// TwinCAT 3 PLC project Nepionic_Motion
// Title: Nepionic_Motion
// Company: Nepionic
// Author: Nepionic
// ProjectVersion: 0.1.0
// ProgramVersion: 3.1.4026.19
// libraries:
//   Nepionic_Core, * (Nepionic)
//   Tc2_MC2, * (Beckhoff Automation GmbH)
//   Tc2_MC2_Drive, * (Beckhoff Automation GmbH)
// project tree:
//   Builders/Homing/ HomeBuilder.TcIO, PositionHomeBuilder.TcIO
//   Builders/Homing/Implementation/ DefaultPositionHomeBuilder.TcPOU, DefaultHomeBuilder.TcPOU, DefaultHomeBuilderParameters.TcDUT
//   Builders/Motion/ GearInBuilder.TcIO (not stored), MotionBuilder.TcIO, AbsoluteMoveBuilder.TcIO, MoveBuilder.TcIO, RelativeMoveBuilder.TcIO, VelocityMoveBuilder.TcIO
//   Builders/Motion/Implementation/ DefaultMotionBuilderParameters.TcDUT, DefaultGearInBuilder.TcPOU, DefaultMotionBuilder.TcPOU, DefaultAbsoluteMoveBuilder.TcPOU, DefaultMoveBuilder.TcPOU, DefaultRelativeMoveBuilder.TcPOU, DefaultVelocityMoveBuilder.TcPOU
//   Commands/Administrative/ ResetCommand.TcPOU (not stored)
//   Commands/Homing/ HomeCommand.TcPOU
//   Commands/SoE/ ResetSoeDriveCommand.TcPOU
//   Commands/Coupling/ GearInCommand.TcPOU, GearOutCommand.TcPOU (not stored)
//   Commands/PointToPoint/ MoveAbsoluteCommand.TcPOU, MoveAdditiveCommand.TcPOU, MoveContinuousAbsoluteCommand.TcPOU, MoveContinuousRelativeCommand.TcPOU, MoveModuloCommand.TcPOU, MoveRelativeCommand.TcPOU, MoveVelocityCommand.TcPOU
//   Commands/Stops/ HaltCommand.TcPOU, StopCommand.TcPOU
//   Command/ Mc2Command.TcPOU, Mc2MotionCommand.TcPOU, MotionCommand.TcIO
//   Functions/ Mc2BufferModeConvertFrom.TcPOU, Mc2BufferModeConvertTo.TcPOU, Mc2DirectionConvertFrom.TcPOU, Mc2DirectionConvertTo.TcPOU, Mc2EncoderReferenceModeConvertFrom.TcPOU, Mc2EncoderReferenceModeConvertTo.TcPOU, Mc2HomingModeConvertFrom.TcPOU, Mc2HomingModeConvertTo.TcPOU
//   Axis/ Axis.TcIO, Mc2Axis.TcPOU
//   Types/ AxisMotionState.TcDUT (not stored), EncoderReferenceMode.TcDUT, HomingMode.TcDUT, MotionBufferMode.TcDUT, MotionDirection.TcDUT

// ---- Builders/Homing/Implementation/DefaultHomeBuilderParameters.TcDUT
TYPE DefaultHomeBuilderParameters :
STRUCT
	position : LREAL;
	homing_mode : HomingMode;
	reference_mode : EncoderReferenceMode;
	search_direction : MotionDirection;
	search_velocity : LREAL;
	sync_direction : MotionDirection;
	sync_velocity : LREAL;
	buffer_mode : MotionBufferMode;
END_STRUCT
END_TYPE

// ---- Builders/Motion/Implementation/DefaultMotionBuilderParameters.TcDUT
TYPE DefaultMotionBuilderParameters :
STRUCT
	position : LREAL;
	distance : LREAL;
	velocity : LREAL;
	acceleration : LREAL;
	deceleration : LREAL;
	jerk : LREAL;
	buffer_mode : MotionBufferMode;
	ratio_numerator : LREAL;
	ratio_denominator : UINT;
END_STRUCT
END_TYPE

// ---- Types/EncoderReferenceMode.TcDUT
{attribute 'qualified_only'}
{attribute 'strict'}
{attribute 'to_string'}
TYPE EncoderReferenceMode :
(
    Default := TO_INT(EncoderReferenceMode_Default),
    PlcCam := TO_INT(EncoderReferenceMode_PlcCam),
    HardwareSync := TO_INT(EncoderReferenceMode_HardwareSync),
    HardwareLatchPositive := TO_INT(EncoderReferenceMode_HardwareLatchPos),
    HardwareLatchNegative := TO_INT(EncoderReferenceMode_HardwareLatchNeg),
    SoftwareSync := TO_INT(EncoderReferenceMode_SoftwareSync),
    SoftDriveLatchPositive := TO_INT(EncoderReferenceMode_SoftDriveLatchPos),
    SoftDriveLatchNegative := TO_INT(EncoderReferenceMode_SoftDriveLatchNeg)
);
END_TYPE

// ---- Types/HomingMode.TcDUT
{attribute 'qualified_only'}
{attribute 'strict'}
{attribute 'to_string'}
TYPE HomingMode :
(
	Default := TO_INT(Tc2_Mc2.MC_DefaultHoming),
	Direct := TO_INT(Tc2_Mc2.MC_Direct),
	ForceCalibration := TO_INT(Tc2_Mc2.MC_ForceCalibration),
	ResetCalibration := TO_INT(Tc2_Mc2.MC_ResetCalibration)
);
END_TYPE

// ---- Types/MotionBufferMode.TcDUT
{attribute 'qualified_only'}
{attribute 'strict'}
{attribute 'to_string'}
TYPE MotionBufferMode :
(
	Aborting,
    Buffered,
    BlendingLow,
    BlendingPrevious,
    BlendingNext,
    BlendingHigh
);
END_TYPE

// ---- Types/MotionDirection.TcDUT
{attribute 'qualified_only'}
{attribute 'strict'}
{attribute 'to_string'}
TYPE MotionDirection :
(
    Positive,
    ShortestWay,
    Negative,
    Current,
    Undefined
);
END_TYPE

// ---- Builders/Homing/HomeBuilder.TcIO
INTERFACE PUBLIC HomeBuilder EXTENDS __System.IQueryInterface

METHOD PUBLIC BufferMode : HomeBuilder
VAR_INPUT
	value : MotionBufferMode;
END_VAR
END_METHOD

METHOD PUBLIC BuildDefaultHomingCommand : AsyncCommand
VAR_INPUT
	axis : Axis;
END_VAR
END_METHOD

METHOD PUBLIC BuildDirectCommand : AsyncCommand
VAR_INPUT
	axis : Axis;
END_VAR
END_METHOD

METHOD PUBLIC BuildForceCalibrationCommand : AsyncCommand
VAR_INPUT
	axis : Axis;
END_VAR
END_METHOD

METHOD PUBLIC BuildResetCalibrationCommand : AsyncCommand
VAR_INPUT
	axis : Axis;
END_VAR
END_METHOD

METHOD PUBLIC Position : PositionHomeBuilder
VAR_INPUT
	value : LREAL;
END_VAR
END_METHOD

METHOD PUBLIC Reset : HomeBuilder
END_METHOD

METHOD PUBLIC SearchDirection : HomeBuilder
VAR_INPUT
	value : MotionDirection;
END_VAR
END_METHOD

METHOD PUBLIC SearchVelocity : HomeBuilder
VAR_INPUT
	value : LREAL;
END_VAR
END_METHOD

METHOD PUBLIC SyncDirection : HomeBuilder
VAR_INPUT
	value : MotionDirection;
END_VAR
END_METHOD

METHOD PUBLIC SyncVelocity : HomeBuilder
VAR_INPUT
	value : LREAL;
END_VAR
END_METHOD

END_INTERFACE

// ---- Builders/Homing/PositionHomeBuilder.TcIO
INTERFACE PUBLIC PositionHomeBuilder EXTENDS __System.IQueryInterface

METHOD PUBLIC BufferMode : PositionHomeBuilder
VAR_INPUT
	value : MotionBufferMode;
END_VAR
END_METHOD

METHOD PUBLIC BuildDefaultHomingCommand : AsyncCommand
VAR_INPUT
	axis : Axis;
END_VAR
END_METHOD

METHOD PUBLIC BuildDirectCommand : AsyncCommand
VAR_INPUT
	axis : Axis;
END_VAR
END_METHOD

METHOD PUBLIC Position : PositionHomeBuilder
VAR_INPUT
	value : LREAL;
END_VAR
END_METHOD

METHOD PUBLIC Reset : PositionHomeBuilder
END_METHOD

METHOD PUBLIC SearchDirection : PositionHomeBuilder
VAR_INPUT
	value : MotionDirection;
END_VAR
END_METHOD

METHOD PUBLIC SearchVelocity : PositionHomeBuilder
VAR_INPUT
	value : LREAL;
END_VAR
END_METHOD

METHOD PUBLIC SyncDirection : PositionHomeBuilder
VAR_INPUT
	value : MotionDirection;
END_VAR
END_METHOD

METHOD PUBLIC SyncVelocity : PositionHomeBuilder
VAR_INPUT
	value : LREAL;
END_VAR
END_METHOD

END_INTERFACE

// ---- Builders/Motion/MotionBuilder.TcIO
INTERFACE PUBLIC MotionBuilder EXTENDS __System.IQueryInterface

METHOD PUBLIC Acceleration : MoveBuilder
VAR_INPUT
	value : LREAL;
END_VAR
END_METHOD

METHOD PUBLIC BufferMode : MoveBuilder
VAR_INPUT
	mode : MotionBufferMode;
END_VAR
END_METHOD

METHOD PUBLIC BuildGearOutCommand : AsyncCommand
VAR_INPUT
	axis : Axis;
END_VAR
END_METHOD

METHOD PUBLIC BuildHaltCommand : MotionCommand
VAR_INPUT
	axis : Axis;
END_VAR
END_METHOD

METHOD PUBLIC BuildStopCommand : MotionCommand
VAR_INPUT
	axis : Axis;
END_VAR
END_METHOD

METHOD PUBLIC Deceleration : MotionBuilder
VAR_INPUT
	value : LREAL;
END_VAR
END_METHOD

METHOD PUBLIC Denominator : GearInBuilder
VAR_INPUT
	value : UINT;
END_VAR
END_METHOD

METHOD PUBLIC Distance : RelativeMoveBuilder
VAR_INPUT
	value : LREAL;
END_VAR
END_METHOD

METHOD PUBLIC Jerk : MotionBuilder
VAR_INPUT
	value : LREAL;
END_VAR
END_METHOD

METHOD PUBLIC Numerator : GearInBuilder
VAR_INPUT
	value : LREAL;
END_VAR
END_METHOD

METHOD PUBLIC Position : AbsoluteMoveBuilder
VAR_INPUT
	value : LREAL;
END_VAR
END_METHOD

METHOD PUBLIC Reset : MotionBuilder
END_METHOD

METHOD PUBLIC Velocity : VelocityMoveBuilder
VAR_INPUT
	value : LREAL;
END_VAR
END_METHOD

END_INTERFACE

// ---- Builders/Motion/AbsoluteMoveBuilder.TcIO
INTERFACE PUBLIC AbsoluteMoveBuilder EXTENDS __System.IQueryInterface

METHOD PUBLIC Acceleration : AbsoluteMoveBuilder
VAR_INPUT
	value : LREAL;
END_VAR
END_METHOD

METHOD PUBLIC BufferMode : AbsoluteMoveBuilder
VAR_INPUT
	mode : MotionBufferMode;
END_VAR
END_METHOD

METHOD PUBLIC BuildMoveAbsoluteCommand : MotionCommand
VAR_INPUT
	axis : Axis;
END_VAR
END_METHOD

METHOD PUBLIC Deceleration : AbsoluteMoveBuilder
VAR_INPUT
	value : LREAL;
END_VAR
END_METHOD

METHOD PUBLIC Jerk : AbsoluteMoveBuilder
VAR_INPUT
	value : LREAL;
END_VAR
END_METHOD

METHOD PUBLIC Position : AbsoluteMoveBuilder
VAR_INPUT
	value : LREAL;
END_VAR
END_METHOD

METHOD PUBLIC Velocity : AbsoluteMoveBuilder
VAR_INPUT
	value : LREAL;
END_VAR
END_METHOD

END_INTERFACE

// ---- Builders/Motion/MoveBuilder.TcIO
INTERFACE PUBLIC MoveBuilder EXTENDS __System.IQueryInterface

METHOD PUBLIC Acceleration : MoveBuilder
VAR_INPUT
	value : LREAL;
END_VAR
END_METHOD

METHOD PUBLIC BufferMode : MoveBuilder
VAR_INPUT
	mode : MotionBufferMode;
END_VAR
END_METHOD

METHOD PUBLIC BuildHaltCommand : MotionCommand
VAR_INPUT
	axis : Axis;
END_VAR
END_METHOD

METHOD PUBLIC Deceleration : MoveBuilder
VAR_INPUT
	value : LREAL;
END_VAR
END_METHOD

METHOD PUBLIC Denominator : GearInBuilder
VAR_INPUT
	value : UINT;
END_VAR
END_METHOD

METHOD PUBLIC Distance : RelativeMoveBuilder
VAR_INPUT
	value : LREAL;
END_VAR
END_METHOD

METHOD PUBLIC Jerk : MoveBuilder
VAR_INPUT
	value : LREAL;
END_VAR
END_METHOD

METHOD PUBLIC Numerator : GearInBuilder
VAR_INPUT
	value : LREAL;
END_VAR
END_METHOD

METHOD PUBLIC Position : AbsoluteMoveBuilder
VAR_INPUT
	value : LREAL;
END_VAR
END_METHOD

METHOD PUBLIC Reset : MoveBuilder
END_METHOD

METHOD PUBLIC Velocity : VelocityMoveBuilder
VAR_INPUT
	value : LREAL;
END_VAR
END_METHOD

END_INTERFACE

// ---- Builders/Motion/RelativeMoveBuilder.TcIO
INTERFACE PUBLIC RelativeMoveBuilder EXTENDS __System.IQueryInterface

METHOD PUBLIC Acceleration : RelativeMoveBuilder
VAR_INPUT
	value : LREAL;
END_VAR
END_METHOD

METHOD PUBLIC BufferMode : RelativeMoveBuilder
VAR_INPUT
	mode : MotionBufferMode;
END_VAR
END_METHOD

METHOD PUBLIC BuildMoveAdditiveCommand : MotionCommand
VAR_INPUT
	axis : Axis;
END_VAR
END_METHOD

METHOD PUBLIC BuildMoveRelativeCommand : MotionCommand
VAR_INPUT
	axis : Axis;
END_VAR
END_METHOD

METHOD PUBLIC Deceleration : RelativeMoveBuilder
VAR_INPUT
	value : LREAL;
END_VAR
END_METHOD

METHOD PUBLIC Distance : RelativeMoveBuilder
VAR_INPUT
	value : LREAL;
END_VAR
END_METHOD

METHOD PUBLIC Jerk : RelativeMoveBuilder
VAR_INPUT
	value : LREAL;
END_VAR
END_METHOD

METHOD PUBLIC Velocity : RelativeMoveBuilder
VAR_INPUT
	value : LREAL;
END_VAR
END_METHOD

END_INTERFACE

// ---- Builders/Motion/VelocityMoveBuilder.TcIO
INTERFACE PUBLIC VelocityMoveBuilder EXTENDS __System.IQueryInterface

METHOD PUBLIC Acceleration : VelocityMoveBuilder
VAR_INPUT
	value : LREAL;
END_VAR
END_METHOD

METHOD PUBLIC BufferMode : VelocityMoveBuilder
VAR_INPUT
	mode : MotionBufferMode;
END_VAR
END_METHOD

METHOD PUBLIC BuildMoveVelocityCommand : MotionCommand
VAR_INPUT
	axis : Axis;
END_VAR
END_METHOD

METHOD PUBLIC Deceleration : VelocityMoveBuilder
VAR_INPUT
	value : LREAL;
END_VAR
END_METHOD

METHOD PUBLIC Distance : RelativeMoveBuilder
VAR_INPUT
	value : LREAL;
END_VAR
END_METHOD

METHOD PUBLIC Jerk : VelocityMoveBuilder
VAR_INPUT
	value : LREAL;
END_VAR
END_METHOD

METHOD PUBLIC Position : AbsoluteMoveBuilder
VAR_INPUT
	value : LREAL;
END_VAR
END_METHOD

METHOD PUBLIC Velocity : VelocityMoveBuilder
VAR_INPUT
	value : LREAL;
END_VAR
END_METHOD

END_INTERFACE

// ---- Command/MotionCommand.TcIO
INTERFACE PUBLIC MotionCommand EXTENDS AsyncCommand

{attribute 'monitoring' := 'call'}
PROPERTY PUBLIC Active : BOOL
GET
END_GET
END_PROPERTY

END_INTERFACE

// ---- Axis/Axis.TcIO
INTERFACE PUBLIC Axis EXTENDS __System.IQueryInterface

{attribute 'monitoring' := 'call'}
PROPERTY PUBLIC ActualAcceleration : LREAL
GET
END_GET
END_PROPERTY

{attribute 'monitoring' := 'call'}
PROPERTY PUBLIC ActualPosition : LREAL
GET
END_GET
END_PROPERTY

{attribute 'monitoring' := 'call'}
PROPERTY PUBLIC ActualVelocity : LREAL
GET
END_GET
END_PROPERTY

PROPERTY PUBLIC AxisRef : REFERENCE TO Tc2_Mc2.Axis_Ref
GET
END_GET
END_PROPERTY

METHOD PUBLIC Disable
END_METHOD

METHOD PUBLIC DisableNegative
END_METHOD

METHOD PUBLIC DisablePositive
END_METHOD

METHOD PUBLIC Enable
END_METHOD

METHOD PUBLIC EnableNegative
END_METHOD

METHOD PUBLIC EnablePositive
END_METHOD

{attribute 'monitoring' := 'call'}
PROPERTY PUBLIC ErrorId : UDINT
GET
END_GET
END_PROPERTY

{attribute 'monitoring' := 'call'}
PROPERTY PUBLIC HasBeenStopped : BOOL
GET
END_GET
END_PROPERTY

{attribute 'monitoring' := 'call'}
PROPERTY PUBLIC HasJob : BOOL
GET
END_GET
END_PROPERTY

{attribute 'monitoring' := 'call'}
PROPERTY PUBLIC IsAccelerating : BOOL
GET
END_GET
END_PROPERTY

{attribute 'monitoring' := 'call'}
PROPERTY PUBLIC IsBusyHoming : BOOL
GET
END_GET
END_PROPERTY

{attribute 'monitoring' := 'call'}
PROPERTY PUBLIC IsCamDataQueued : BOOL
GET
END_GET
END_PROPERTY

{attribute 'monitoring' := 'call'}
PROPERTY PUBLIC IsCamScalingPending : BOOL
GET
END_GET
END_PROPERTY

{attribute 'monitoring' := 'call'}
PROPERTY PUBLIC IsCamTableQueued : BOOL
GET
END_GET
END_PROPERTY

{attribute 'monitoring' := 'call'}
PROPERTY PUBLIC IsCommandBuffered : BOOL
GET
END_GET
END_PROPERTY

{attribute 'monitoring' := 'call'}
PROPERTY PUBLIC IsCompensating : BOOL
GET
END_GET
END_PROPERTY

{attribute 'monitoring' := 'call'}
PROPERTY PUBLIC IsConstantVelocity : BOOL
GET
END_GET
END_PROPERTY

{attribute 'monitoring' := 'call'}
PROPERTY PUBLIC IsContinuousMotion : BOOL
GET
END_GET
END_PROPERTY

{attribute 'monitoring' := 'call'}
PROPERTY PUBLIC IsControlLoopClosed : BOOL
GET
END_GET
END_PROPERTY

{attribute 'monitoring' := 'call'}
PROPERTY PUBLIC IsCoupled : BOOL
GET
END_GET
END_PROPERTY

{attribute 'monitoring' := 'call'}
PROPERTY PUBLIC IsDecelerating : BOOL
GET
END_GET
END_PROPERTY

{attribute 'monitoring' := 'call'}
PROPERTY PUBLIC IsDisabled : BOOL
GET
END_GET
END_PROPERTY

{attribute 'monitoring' := 'call'}
PROPERTY PUBLIC IsDiscreteMotion : BOOL
GET
END_GET
END_PROPERTY

{attribute 'monitoring' := 'call'}
PROPERTY PUBLIC IsDriveDeviceErrored : BOOL
GET
END_GET
END_PROPERTY

{attribute 'monitoring' := 'call'}
PROPERTY PUBLIC IsErrored : BOOL
GET
END_GET
END_PROPERTY

{attribute 'monitoring' := 'call'}
PROPERTY PUBLIC IsErrorStop : BOOL
GET
END_GET
END_PROPERTY

{attribute 'monitoring' := 'call'}
PROPERTY PUBLIC IsExternalLatchValid : BOOL
GET
END_GET
END_PROPERTY

{attribute 'monitoring' := 'call'}
PROPERTY PUBLIC IsExtSetPointGenEnabled : BOOL
GET
END_GET
END_PROPERTY

{attribute 'monitoring' := 'call'}
PROPERTY PUBLIC IsHomed : BOOL
GET
END_GET
END_PROPERTY

{attribute 'monitoring' := 'call'}
PROPERTY PUBLIC IsHoming : BOOL
GET
END_GET
END_PROPERTY

{attribute 'monitoring' := 'call'}
PROPERTY PUBLIC IsInPositionArea : BOOL
GET
END_GET
END_PROPERTY

{attribute 'monitoring' := 'call'}
PROPERTY PUBLIC IsInTargetPosition : BOOL
GET
END_GET
END_PROPERTY

{attribute 'monitoring' := 'call'}
PROPERTY PUBLIC IsIoDataInvalid : BOOL
GET
END_GET
END_PROPERTY

{attribute 'monitoring' := 'call'}
PROPERTY PUBLIC IsMotionCommandsLocked : BOOL
GET
END_GET
END_PROPERTY

{attribute 'monitoring' := 'call'}
PROPERTY PUBLIC IsMoving : BOOL
GET
END_GET
END_PROPERTY

{attribute 'monitoring' := 'call'}
PROPERTY PUBLIC IsNegativeDirection : BOOL
GET
END_GET
END_PROPERTY

{attribute 'monitoring' := 'call'}
PROPERTY PUBLIC IsNewTargetPosition : BOOL
GET
END_GET
END_PROPERTY

{attribute 'monitoring' := 'call'}
PROPERTY PUBLIC IsNotMoving : BOOL
GET
END_GET
END_PROPERTY

{attribute 'monitoring' := 'call'}
PROPERTY PUBLIC IsOperational : BOOL
GET
END_GET
END_PROPERTY

{attribute 'monitoring' := 'call'}
PROPERTY PUBLIC IsPointToPointMode : BOOL
GET
END_GET
END_PROPERTY

{attribute 'monitoring' := 'call'}
PROPERTY PUBLIC IsPositiveDirection : BOOL
GET
END_GET
END_PROPERTY

{attribute 'monitoring' := 'call'}
PROPERTY PUBLIC IsProtected : BOOL
GET
END_GET
END_PROPERTY

{attribute 'monitoring' := 'call'}
PROPERTY PUBLIC IsSoftLimitMaxExceeded : BOOL
GET
END_GET
END_PROPERTY

{attribute 'monitoring' := 'call'}
PROPERTY PUBLIC IsSoftLimitMinExceeded : BOOL
GET
END_GET
END_PROPERTY

{attribute 'monitoring' := 'call'}
PROPERTY PUBLIC IsStandstill : BOOL
GET
END_GET
END_PROPERTY

{attribute 'monitoring' := 'call'}
PROPERTY PUBLIC IsStopping : BOOL
GET
END_GET
END_PROPERTY

{attribute 'monitoring' := 'call'}
PROPERTY PUBLIC IsSynchronisedMotion : BOOL
GET
END_GET
END_PROPERTY

{attribute 'monitoring' := 'call'}
PROPERTY PUBLIC MotionState : AxisMotionState
GET
END_GET
END_PROPERTY

PROPERTY PUBLIC OpMode : Tc2_Mc2.St_AxisOpModes
GET
END_GET
END_PROPERTY

PROPERTY PUBLIC Override : LREAL
GET
END_GET
SET
END_SET
END_PROPERTY

METHOD PUBLIC Reset : AsyncCommand
END_METHOD

METHOD PUBLIC ResetDrive : AsyncCommand
END_METHOD

METHOD PUBLIC SetPosition : AsyncCommand
VAR_INPUT
	position : LREAL;
END_VAR
END_METHOD

{attribute 'monitoring' := 'call'}
PROPERTY PUBLIC TargetPosition : LREAL
GET
END_GET
END_PROPERTY

END_INTERFACE

// ---- Builders/Homing/Implementation/DefaultPositionHomeBuilder.TcPOU
{attribute 'linkalways'} 
{attribute 'no_explicit_call' := 'This FB is a CLASS and must be accessed using methods or properties'}
{attribute 'enable_dynamic_creation'}
FUNCTION_BLOCK PUBLIC DefaultPositionHomeBuilder IMPLEMENTS PositionHomeBuilder
VAR
	parent_builder : POINTER TO DefaultHomeBuilder;
END_VAR

METHOD PUBLIC BufferMode : PositionHomeBuilder
VAR_INPUT
	value : MotionBufferMode;
END_VAR
parent_builder^.BufferMode(value);
BufferMode := THIS^;
END_METHOD

METHOD PUBLIC BuildDefaultHomingCommand : AsyncCommand
VAR_INPUT
	axis : Axis;
END_VAR
BuildDefaultHomingCommand := parent_builder^.BuildDefaultHomingCommand(axis);
END_METHOD

METHOD PUBLIC BuildDirectCommand : AsyncCommand
VAR_INPUT
	axis : Axis;
END_VAR
BuildDirectCommand := parent_builder^.BuildDirectCommand(axis);
END_METHOD

//FB_Init is always available implicitly and it is used primarily for initialization.
//The return value is not evaluated. For a specific influence, you can also declare the
//methods explicitly and provide additional code there with the standard initialization
//code. You can evaluate the return value.
METHOD FB_Init: BOOL
VAR_INPUT
    bInitRetains : BOOL; // TRUE: the retain variables are initialized (reset warm / reset cold)
    bInCopyCode : BOOL;  // TRUE: the instance will be copied to the copy code afterward (online change)
	parent_builder : POINTER TO DefaultHomeBuilder;
END_VAR
THIS^.parent_builder := parent_builder;
END_METHOD

METHOD PUBLIC Position : PositionHomeBuilder
VAR_INPUT
	value : LREAL;
END_VAR
parent_builder^.Position(value);
Position := THIS^;
END_METHOD

METHOD PUBLIC Reset : PositionHomeBuilder
parent_builder^.Reset();
Reset := THIS^;
END_METHOD

METHOD PUBLIC SearchDirection : PositionHomeBuilder
VAR_INPUT
	value : MotionDirection;
END_VAR
parent_builder^.SearchDirection(value);
SearchDirection := THIS^;
END_METHOD

METHOD PUBLIC SearchVelocity : PositionHomeBuilder
VAR_INPUT
	value : LREAL;
END_VAR
parent_builder^.SearchVelocity(value);
SearchVelocity := THIS^;
END_METHOD

METHOD PUBLIC SyncDirection : PositionHomeBuilder
VAR_INPUT
	value : MotionDirection;
END_VAR
parent_builder^.SyncDirection(value);
SyncDirection := THIS^;
END_METHOD

METHOD PUBLIC SyncVelocity : PositionHomeBuilder
VAR_INPUT
	value : LREAL;
END_VAR
parent_builder^.SyncVelocity(value);
SyncVelocity := THIS^;
END_METHOD

END_FUNCTION_BLOCK

// ---- Builders/Homing/Implementation/DefaultHomeBuilder.TcPOU
{attribute 'linkalways'} 
{attribute 'no_explicit_call' := 'This FB is a CLASS and must be accessed using methods or properties'}
{attribute 'enable_dynamic_creation'}
FUNCTION_BLOCK PUBLIC DefaultHomeBuilder IMPLEMENTS HomeBuilder
VAR
	parameters : DefaultHomeBuilderParameters;
	position_home_builder : DefaultPositionHomeBuilder(parent_builder := THIS);
END_VAR
VAR CONSTANT
	default_parameters : DefaultHomeBuilderParameters := (
		homing_mode := HomingMode.Default,
		reference_mode := EncoderReferenceMode.Default,
		search_direction := MotionDirection.Positive,
		search_velocity := 0,
		sync_direction := MotionDirection.Positive,
		sync_velocity := 0,
		buffer_mode := MotionBufferMode.Aborting
	);	
END_VAR

METHOD PUBLIC BufferMode : HomeBuilder
VAR_INPUT
	value : MotionBufferMode;
END_VAR
parameters.buffer_mode := value;
BufferMode := THIS^;
END_METHOD

METHOD PUBLIC BuildDefaultHomingCommand : AsyncCommand
VAR_INPUT
	axis : Axis;
END_VAR
VAR
	command_ptr : POINTER TO HomeCommand;
	command : AsyncCommand;
END_VAR
command_ptr := __NEW(HomeCommand(
	axis := axis,
	position := parameters.position,
	homing_mode := HomingMode.Default,
 	buffer_mode := parameters.buffer_mode
));
BuildDefaultHomingCommand := command_ptr^;
END_METHOD

METHOD PUBLIC BuildDirectCommand : AsyncCommand
VAR_INPUT
	axis : Axis;
END_VAR
VAR
	command_ptr : POINTER TO HomeCommand;
	command : AsyncCommand;
END_VAR
command_ptr := __NEW(HomeCommand(
	axis := axis,
	position := parameters.position,
	homing_mode := HomingMode.Direct,
 	buffer_mode := parameters.buffer_mode
));
BuildDirectCommand := command_ptr^;
END_METHOD

METHOD PUBLIC BuildForceCalibrationCommand : AsyncCommand
VAR_INPUT
	axis : Axis;
END_VAR
VAR
	command_ptr : POINTER TO HomeCommand;
	command : AsyncCommand;
END_VAR
command_ptr := __NEW(HomeCommand(
	axis := axis,
	position := parameters.position,
	homing_mode := HomingMode.ForceCalibration,
 	buffer_mode := parameters.buffer_mode
));
BuildForceCalibrationCommand := command_ptr^;
END_METHOD

METHOD PUBLIC BuildResetCalibrationCommand : AsyncCommand
VAR_INPUT
	axis : Axis;
END_VAR
VAR
	command_ptr : POINTER TO HomeCommand;
	command : AsyncCommand;
END_VAR
command_ptr := __NEW(HomeCommand(
	axis := axis,
	position := 0,
	homing_mode := HomingMode.ResetCalibration,
 	buffer_mode := parameters.buffer_mode
));
BuildResetCalibrationCommand := command_ptr^;
END_METHOD

METHOD PUBLIC Position : PositionHomeBuilder
VAR_INPUT
	value : LREAL;
END_VAR
parameters.position := value;
Position := position_home_builder;
END_METHOD

METHOD PUBLIC Reset : HomeBuilder
parameters := default_parameters;
Reset := THIS^;
END_METHOD

METHOD PUBLIC SearchDirection : HomeBuilder
VAR_INPUT
	value : MotionDirection;
END_VAR
parameters.search_direction := value;
SearchDirection := THIS^;
END_METHOD

METHOD PUBLIC SearchVelocity : HomeBuilder
VAR_INPUT
	value : LREAL;
END_VAR
parameters.search_velocity := value;
SearchVelocity := THIS^;
END_METHOD

METHOD PUBLIC SyncDirection : HomeBuilder
VAR_INPUT
	value : MotionDirection;
END_VAR
parameters.sync_direction := value;
SyncDirection := THIS^;
END_METHOD

METHOD PUBLIC SyncVelocity : HomeBuilder
VAR_INPUT
	value : LREAL;
END_VAR
parameters.sync_velocity := value;
SyncVelocity := THIS^;
END_METHOD

END_FUNCTION_BLOCK

// ---- Commands/Homing/HomeCommand.TcPOU
{attribute 'linkalways'} 
{attribute 'no_explicit_call' := 'This FB is a CLASS and must be accessed using methods or properties'}
{attribute 'enable_dynamic_creation'}
FUNCTION_BLOCK HomeCommand EXTENDS Mc2Command
VAR
	fb : Tc2_Mc2.Mc_Home;
END_VAR

METHOD PUBLIC CyclicCall
SUPER^.CyclicCall();
fb(Axis := axis_ref);
END_METHOD

(*FB_Init is always available implicitly and it is used primarily for initialization.
The return value is not evaluated. For a specific influence, you can also declare the
methods explicitly and provide additional code there with the standard initialization
code. You can evaluate the return value.*)
METHOD FB_Init : BOOL
VAR_INPUT
	(* TRUE: the retain variables are initialized (reset warm / reset cold)*)
	bInitRetains : BOOL;
	(* TRUE: the instance will be copied to the copy code afterward (online change)*)
	bInCopyCode	: BOOL;
	axis : Axis;
	position : LREAL := Tc2_Mc2.Default_Home_Position;
	homing_mode : HomingMode := HomingMode.Default;
	buffer_mode	: MotionBufferMode := MotionBufferMode.Aborting;
END_VAR
fb.Position := position;
fb.HomingMode := Mc2HomingModeConvertTo(homing_mode);
fb.BufferMode := Mc2BufferModeConvertTo(buffer_mode);
END_METHOD

METHOD PROTECTED OnExecuting
VAR_INPUT
	state_control : AsyncCommandStateControl;
END_VAR
fb.Execute := TRUE;

IF fb.Done THEN
	state_control.Next();
	fb.Execute := FALSE;
END_IF

IF fb.CommandAborted THEN
	Abort();
	fb.Execute := FALSE;
END_IF

IF fb.Error THEN
	state_control.Error(fb.ErrorId);
	fb.Execute := FALSE;
END_IF
END_METHOD

END_FUNCTION_BLOCK

// ---- Command/Mc2Command.TcPOU
{attribute 'linkalways'} 
{attribute 'no_explicit_call' := 'This FB is a CLASS and must be accessed using methods or properties'}
{attribute 'enable_dynamic_creation'}
FUNCTION_BLOCK PUBLIC ABSTRACT Mc2Command EXTENDS NoopAsyncCommand IMPLEMENTS AsyncCommand
VAR
	axis_ref : REFERENCE TO Tc2_Mc2.Axis_Ref;
END_VAR

//FB_Init is always available implicitly and it is used primarily for initialization.
//The return value is not evaluated. For a specific influence, you can also declare the
//methods explicitly and provide additional code there with the standard initialization
//code. You can evaluate the return value.
METHOD FB_Init: BOOL
VAR_INPUT
    bInitRetains: BOOL; // TRUE: the retain variables are initialized (reset warm / reset cold)
    bInCopyCode: BOOL;  // TRUE: the instance will be copied to the copy code afterward (online change)
	axis : Axis;   
END_VAR
axis_ref REF= axis.AxisRef;
END_METHOD

METHOD PROTECTED ABSTRACT OnExecuting
VAR_INPUT
	state_control : AsyncCommandStateControl;
END_VAR
END_METHOD

END_FUNCTION_BLOCK

// ---- Functions/Mc2HomingModeConvertTo.TcPOU
FUNCTION Mc2HomingModeConvertTo : Tc2_Mc2.Mc_HomingMode
VAR_INPUT
	homing_mode : HomingMode;
END_VAR

CASE homing_mode OF
	HomingMode.Default: Mc2HomingModeConvertTo := Tc2_Mc2.MC_DefaultHoming;
	HomingMode.Direct: Mc2HomingModeConvertTo := Tc2_Mc2.MC_Direct;
	HomingMode.ForceCalibration: Mc2HomingModeConvertTo := Tc2_Mc2.MC_ForceCalibration;
	HomingMode.ResetCalibration: Mc2HomingModeConvertTo := Tc2_Mc2.MC_ResetCalibration;
END_CASE

END_FUNCTION

// ---- Functions/Mc2BufferModeConvertTo.TcPOU
FUNCTION INTERNAL Mc2BufferModeConvertTo : Tc2_Mc2.Mc_BufferMode
VAR_INPUT
	buffer_mode : MotionBufferMode;
END_VAR

CASE buffer_mode OF
	MotionBufferMode.Aborting: Mc2BufferModeConvertTo := Tc2_Mc2.Mc_BufferMode.Mc_Aborting;
    MotionBufferMode.Buffered: Mc2BufferModeConvertTo := Tc2_Mc2.Mc_BufferMode.Mc_Buffered;
    MotionBufferMode.BlendingLow: Mc2BufferModeConvertTo := Tc2_Mc2.Mc_BufferMode.Mc_BlendingLow;
   	MotionBufferMode.BlendingPrevious: Mc2BufferModeConvertTo := Tc2_Mc2.Mc_BufferMode.Mc_BlendingPrevious;
    MotionBufferMode.BlendingNext: Mc2BufferModeConvertTo := Tc2_Mc2.Mc_BufferMode.Mc_BlendingNext;
    MotionBufferMode.BlendingHigh: Mc2BufferModeConvertTo := Tc2_Mc2.Mc_BufferMode.Mc_BlendingHigh;
END_CASE

END_FUNCTION

// ---- Builders/Motion/Implementation/DefaultGearInBuilder.TcPOU
{attribute 'linkalways'} 
{attribute 'no_explicit_call' := 'This FB is a CLASS and must be accessed using methods or properties'}
{attribute 'enable_dynamic_creation'}
FUNCTION_BLOCK PUBLIC DefaultGearInBuilder IMPLEMENTS GearInBuilder
VAR
	parent_builder : POINTER TO DefaultMotionBuilder;
END_VAR

METHOD PUBLIC Acceleration : GearInBuilder
VAR_INPUT
	value : LREAL;
END_VAR
parent_builder^.Acceleration(value);
Acceleration := THIS^;
END_METHOD

METHOD PUBLIC BufferMode : GearInBuilder
VAR_INPUT
	mode : MotionBufferMode;
END_VAR
parent_builder^.BufferMode(mode);
BufferMode := THIS^;
END_METHOD

METHOD PUBLIC BuildGearInCommand : AsyncCommand
VAR_INPUT
	master_axis : Axis;
	slave_axis : Axis;
END_VAR
VAR
	command_ptr : POINTER TO GearInCommand;
	command : AsyncCommand;
END_VAR
command_ptr := __NEW(GearInCommand(
	master_axis := master_axis,
	slave_axis := slave_axis,
	numerator := parent_builder^.Parameters.ratio_numerator,
	denominator := parent_builder^.Parameters.ratio_denominator
// 	deceleration := parameters.deceleration,
// 	jerk := parameters.jerk,
// 	buffer_mode := parameters.buffer_mode
));
BuildGearInCommand := command_ptr^;
END_METHOD

METHOD PUBLIC Deceleration : GearInBuilder
VAR_INPUT
	value : LREAL;
END_VAR
parent_builder^.Deceleration(value);
Deceleration := THIS^;
END_METHOD

METHOD Denominator : GearInBuilder
VAR_INPUT
	value : UINT;
END_VAR
parent_builder^.Denominator(value);
Denominator := THIS^;
END_METHOD

//FB_Init is always available implicitly and it is used primarily for initialization.
//The return value is not evaluated. For a specific influence, you can also declare the
//methods explicitly and provide additional code there with the standard initialization
//code. You can evaluate the return value.
METHOD FB_Init: BOOL
VAR_INPUT
    bInitRetains : BOOL; // TRUE: the retain variables are initialized (reset warm / reset cold)
    bInCopyCode : BOOL;  // TRUE: the instance will be copied to the copy code afterward (online change)
	parent_builder : POINTER TO DefaultMotionBuilder;
END_VAR
THIS^.parent_builder := parent_builder;
END_METHOD

METHOD PUBLIC Jerk : GearInBuilder
VAR_INPUT
	value : LREAL;
END_VAR
parent_builder^.Jerk(value);
Jerk := THIS^;
END_METHOD

METHOD Numerator : GearInBuilder
VAR_INPUT
	value : LREAL;
END_VAR
parent_builder^.Numerator(value);
Numerator := THIS^;
END_METHOD

METHOD PUBLIC Reset : GearInBuilder
parent_builder^.Reset();
Reset := THIS^;
END_METHOD

END_FUNCTION_BLOCK

// ---- Builders/Motion/Implementation/DefaultMotionBuilder.TcPOU
{attribute 'linkalways'} 
{attribute 'no_explicit_call' := 'This FB is a CLASS and must be accessed using methods or properties'}
{attribute 'enable_dynamic_creation'}
FUNCTION_BLOCK PUBLIC DefaultMotionBuilder IMPLEMENTS MotionBuilder
VAR
	_parameters : DefaultMotionBuilderParameters;
	move_builder : DefaultMoveBuilder(parent_builder := THIS);
	velocity_move_builder : DefaultVelocityMoveBuilder(parent_builder := THIS);
	absolute_move_builder : DefaultAbsoluteMoveBuilder(parent_builder := THIS);
	relative_move_builder : DefaultRelativeMoveBuilder(parent_builder := THIS);
	gear_in_builder : DefaultGearInBuilder(parent_builder := THIS);
END_VAR
VAR CONSTANT
	default_parameters : DefaultMotionBuilderParameters := (
		position := 0,
		distance := 0,
		velocity := 0,
		acceleration := 0,
		deceleration := 0,
		jerk := 0,
		buffer_mode := MotionBufferMode.Aborting,
		ratio_numerator := 1,
		ratio_denominator := 1
	);
END_VAR

PROPERTY INTERNAL AbsoluteMoveBuilder : AbsoluteMoveBuilder
GET // INTERNAL
AbsoluteMoveBuilder := absolute_move_builder;
END_GET
END_PROPERTY

METHOD PUBLIC Acceleration : MoveBuilder
VAR_INPUT
	value : LREAL;
END_VAR
_parameters.acceleration := value;
Acceleration := move_builder;
END_METHOD

METHOD PUBLIC BufferMode : MoveBuilder
VAR_INPUT
	mode : MotionBufferMode;
END_VAR
_parameters.buffer_mode := mode;
BufferMode := move_builder;
END_METHOD

METHOD PUBLIC BuildGearOutCommand : AsyncCommand
VAR_INPUT
	axis : Axis;
END_VAR
VAR
	command_ptr : POINTER TO GearOutCommand;
	command : AsyncCommand;
END_VAR
command_ptr := __NEW(GearOutCommand(
	axis := axis
));
BuildGearOutCommand := command_ptr^;
END_METHOD

METHOD PUBLIC BuildHaltCommand : MotionCommand
VAR_INPUT
	axis : Axis;
END_VAR
VAR
	command_ptr : POINTER TO HaltCommand;
	command : MotionCommand;
END_VAR
command_ptr := __NEW(HaltCommand(
	axis := axis,
	deceleration := _parameters.deceleration,
	jerk := _parameters.jerk,
	buffer_mode := _parameters.buffer_mode
));
BuildHaltCommand := command_ptr^;
END_METHOD

METHOD PUBLIC BuildStopCommand : MotionCommand
VAR_INPUT
	axis : Axis;
END_VAR
VAR
	command_ptr : POINTER TO StopCommand;
	command : MotionCommand;
END_VAR
command_ptr := __NEW(StopCommand(
	axis := axis,
	deceleration := _parameters.deceleration,
	jerk := _parameters.jerk
));
BuildStopCommand := command_ptr^;
END_METHOD

METHOD PUBLIC Deceleration : MotionBuilder
VAR_INPUT
	value : LREAL;
END_VAR
_parameters.deceleration := value;
Deceleration := THIS^;
END_METHOD

METHOD PUBLIC Denominator : GearInBuilder
VAR_INPUT
	value : UINT;
END_VAR
_parameters.ratio_denominator := value;
Denominator := gear_in_builder;
END_METHOD

METHOD PUBLIC Distance : RelativeMoveBuilder
VAR_INPUT
	value : LREAL;
END_VAR
_parameters.distance := value;
Distance := relative_move_builder;
END_METHOD

PROPERTY INTERNAL GearInBuilder : GearInBuilder
GET // INTERNAL
GearInBuilder := gear_in_builder;
END_GET
END_PROPERTY

METHOD PUBLIC Jerk : MotionBuilder
VAR_INPUT
	value : LREAL;
END_VAR
_parameters.jerk := value;
Jerk := THIS^;
END_METHOD

PROPERTY INTERNAL MoveBuilder : MoveBuilder
GET // INTERNAL
MoveBuilder := move_builder;
END_GET
END_PROPERTY

METHOD PUBLIC Numerator : GearInBuilder
VAR_INPUT
	value : LREAL;
END_VAR
_parameters.ratio_numerator := value;
Numerator := gear_in_builder;
END_METHOD

PROPERTY INTERNAL Parameters : REFERENCE TO DefaultMotionBuilderParameters
GET // INTERNAL
Parameters REF= _parameters;
END_GET
END_PROPERTY

METHOD PUBLIC Position : AbsoluteMoveBuilder
VAR_INPUT
	value : LREAL;
END_VAR
_parameters.position := value;
Position := absolute_move_builder;
END_METHOD

PROPERTY INTERNAL RelativeMoveBuilder : RelativeMoveBuilder
GET // INTERNAL
RelativeMoveBuilder := relative_move_builder;
END_GET
END_PROPERTY

METHOD PUBLIC Reset : MotionBuilder
parameters := default_parameters;
Reset := THIS^;
END_METHOD

METHOD PUBLIC Velocity : VelocityMoveBuilder
VAR_INPUT
	value : LREAL;
END_VAR
_parameters.velocity := value;
Velocity := velocity_move_builder;
END_METHOD

PROPERTY INTERNAL VelocityMoveBuilder : VelocityMoveBuilder
GET // INTERNAL
VelocityMoveBuilder := velocity_move_builder;
END_GET
END_PROPERTY

END_FUNCTION_BLOCK

// ---- Builders/Motion/Implementation/DefaultMoveBuilder.TcPOU
{attribute 'linkalways'} 
{attribute 'no_explicit_call' := 'This FB is a CLASS and must be accessed using methods or properties'}
{attribute 'enable_dynamic_creation'}
FUNCTION_BLOCK INTERNAL DefaultMoveBuilder IMPLEMENTS MoveBuilder
VAR
	parent_builder : POINTER TO DefaultMotionBuilder;
END_VAR

METHOD PUBLIC Acceleration : MoveBuilder
VAR_INPUT
	value : LREAL;
END_VAR
parent_builder^.Acceleration(value);
Acceleration := THIS^;
END_METHOD

METHOD PUBLIC BufferMode : MoveBuilder
VAR_INPUT
	mode : MotionBufferMode;
END_VAR
parent_builder^.BufferMode(mode);
BufferMode := THIS^;
END_METHOD

METHOD PUBLIC BuildHaltCommand : MotionCommand
VAR_INPUT
	axis : Axis;
END_VAR
VAR
	command_ptr : POINTER TO HaltCommand;
	command : MotionCommand;
END_VAR
command_ptr := __NEW(HaltCommand(
	axis := axis,
	deceleration := parent_builder^.Parameters.deceleration,
	jerk := parent_builder^.Parameters.jerk,
	buffer_mode := parent_builder^.Parameters.buffer_mode
));
BuildHaltCommand := command_ptr^;
END_METHOD

METHOD PUBLIC Deceleration : MoveBuilder
VAR_INPUT
	value : LREAL;
END_VAR
parent_builder^.Deceleration(value);
Deceleration := THIS^;
END_METHOD

METHOD PUBLIC Denominator : GearInBuilder
VAR_INPUT
	value : UINT;
END_VAR
parent_builder^.Denominator(value);
Denominator := parent_builder^.GearInBuilder;
END_METHOD

METHOD PUBLIC Distance : RelativeMoveBuilder
VAR_INPUT
	value : LREAL;
END_VAR
parent_builder^.Distance(value);
Distance := parent_builder^.RelativeMoveBuilder;
END_METHOD

//FB_Init is always available implicitly and it is used primarily for initialization.
//The return value is not evaluated. For a specific influence, you can also declare the
//methods explicitly and provide additional code there with the standard initialization
//code. You can evaluate the return value.
METHOD FB_Init: BOOL
VAR_INPUT
    bInitRetains : BOOL; // TRUE: the retain variables are initialized (reset warm / reset cold)
    bInCopyCode : BOOL;  // TRUE: the instance will be copied to the copy code afterward (online change)
	parent_builder : POINTER TO DefaultMotionBuilder;
END_VAR
THIS^.parent_builder := parent_builder;
END_METHOD

METHOD PUBLIC Jerk : MoveBuilder
VAR_INPUT
	value : LREAL;
END_VAR
parent_builder^.Jerk(value);
Jerk := THIS^;
END_METHOD

METHOD PUBLIC Numerator : GearInBuilder
VAR_INPUT
	value : LREAL;
END_VAR
parent_builder^.Numerator(value);
Numerator := parent_builder^.GearInBuilder;
END_METHOD

METHOD PUBLIC Position : AbsoluteMoveBuilder
VAR_INPUT
	value : LREAL;
END_VAR
parent_builder^.Position(value);
Position := parent_builder^.AbsoluteMoveBuilder;
END_METHOD

METHOD PUBLIC Reset : MoveBuilder
parent_builder^.Reset();
Reset := THIS^;
END_METHOD

METHOD PUBLIC Velocity : VelocityMoveBuilder
VAR_INPUT
	value : LREAL;
END_VAR
parent_builder^.Velocity(value);
Velocity := parent_builder^.VelocityMoveBuilder;
END_METHOD

END_FUNCTION_BLOCK

// ---- Commands/Stops/HaltCommand.TcPOU
{attribute 'linkalways'} 
{attribute 'no_explicit_call' := 'This FB is a CLASS and must be accessed using methods or properties'}
{attribute 'enable_dynamic_creation'}
FUNCTION_BLOCK HaltCommand EXTENDS Mc2MotionCommand
VAR
	fb : Tc2_Mc2.Mc_Halt;
END_VAR

{attribute 'monitoring' := 'call'}
PROPERTY PUBLIC Active : BOOL
GET // PUBLIC
Active := fb.Active;
END_GET
END_PROPERTY

METHOD PUBLIC CyclicCall
SUPER^.CyclicCall();
fb(Axis := axis_ref);
END_METHOD

(*FB_Init is always available implicitly and it is used primarily for initialization.
The return value is not evaluated. For a specific influence, you can also declare the
methods explicitly and provide additional code there with the standard initialization
code. You can evaluate the return value.*)
METHOD FB_Init : BOOL
VAR_INPUT
	(* TRUE: the retain variables are initialized (reset warm / reset cold)*)
	bInitRetains : BOOL;
	(* TRUE: the instance will be copied to the copy code afterward (online change)*)
	bInCopyCode	: BOOL;
	axis : Axis;
	deceleration : LREAL := 0;
	jerk : LREAL := 0;
	buffer_mode	: MotionBufferMode := MotionBufferMode.Aborting;
END_VAR
fb.Deceleration := deceleration;
fb.Jerk := jerk;
fb.BufferMode := Mc2BufferModeConvertTo(buffer_mode);
END_METHOD

METHOD PROTECTED OnExecuting
VAR_INPUT
	state_control : AsyncCommandStateControl;
END_VAR
fb.Execute := TRUE;

IF fb.Done THEN
	state_control.Next();
	fb.Execute := FALSE;
END_IF

IF fb.CommandAborted THEN
	Abort();
	fb.Execute := FALSE;
END_IF

IF fb.Error THEN
	state_control.Error(fb.ErrorId);
	fb.Execute := FALSE;
END_IF
END_METHOD

END_FUNCTION_BLOCK

// ---- Command/Mc2MotionCommand.TcPOU
{attribute 'linkalways'} 
{attribute 'no_explicit_call' := 'This FB is a CLASS and must be accessed using methods or properties'}
{attribute 'enable_dynamic_creation'}
FUNCTION_BLOCK INTERNAL ABSTRACT Mc2MotionCommand EXTENDS Mc2Command IMPLEMENTS MotionCommand
VAR
END_VAR

{attribute 'monitoring' := 'call'}
PROPERTY PUBLIC ABSTRACT Active : BOOL
GET // PUBLIC
END_GET
END_PROPERTY

END_FUNCTION_BLOCK

// ---- Builders/Motion/Implementation/DefaultVelocityMoveBuilder.TcPOU
{attribute 'linkalways'} 
{attribute 'no_explicit_call' := 'This FB is a CLASS and must be accessed using methods or properties'}
{attribute 'enable_dynamic_creation'}
FUNCTION_BLOCK INTERNAL DefaultVelocityMoveBuilder IMPLEMENTS VelocityMoveBuilder
VAR
	parent_builder : POINTER TO DefaultMotionBuilder;
END_VAR

METHOD PUBLIC Acceleration : VelocityMoveBuilder
VAR_INPUT
	value : LREAL;
END_VAR
parent_builder^.Acceleration(value);
Acceleration := THIS^;
END_METHOD

METHOD PUBLIC BufferMode : VelocityMoveBuilder
VAR_INPUT
	mode : MotionBufferMode;
END_VAR
parent_builder^.BufferMode(mode);
BufferMode := THIS^;
END_METHOD

METHOD PUBLIC BuildMoveVelocityCommand : MotionCommand
VAR_INPUT
	axis : Axis;
END_VAR
VAR
	command_ptr : POINTER TO MoveVelocityCommand;
	command : MotionCommand;
END_VAR
command_ptr := __NEW(MoveVelocityCommand(
	axis := axis,
	velocity := parent_builder^.Parameters.velocity,
	acceleration := parent_builder^.Parameters.acceleration,
	deceleration := parent_builder^.Parameters.deceleration,
	jerk := parent_builder^.Parameters.jerk,
	buffer_mode := parent_builder^.Parameters.buffer_mode
));
BuildMoveVelocityCommand := command_ptr^;
END_METHOD

METHOD PUBLIC Deceleration : VelocityMoveBuilder
VAR_INPUT
	value : LREAL;
END_VAR
parent_builder^.Deceleration(value);
Deceleration := THIS^;
END_METHOD

METHOD PUBLIC Distance : RelativeMoveBuilder
VAR_INPUT
	value : LREAL;
END_VAR
parent_builder^.Distance(value);
Distance := parent_builder^.RelativeMoveBuilder;
END_METHOD

//FB_Init is always available implicitly and it is used primarily for initialization.
//The return value is not evaluated. For a specific influence, you can also declare the
//methods explicitly and provide additional code there with the standard initialization
//code. You can evaluate the return value.
METHOD FB_Init: BOOL
VAR_INPUT
    bInitRetains : BOOL; // TRUE: the retain variables are initialized (reset warm / reset cold)
    bInCopyCode : BOOL;  // TRUE: the instance will be copied to the copy code afterward (online change)
	parent_builder : POINTER TO DefaultMotionBuilder;
END_VAR
THIS^.parent_builder := parent_builder;
END_METHOD

METHOD PUBLIC Jerk : VelocityMoveBuilder
VAR_INPUT
	value : LREAL;
END_VAR
parent_builder^.Jerk(value);
Jerk := THIS^;
END_METHOD

METHOD PUBLIC Position : AbsoluteMoveBuilder
VAR_INPUT
	value : LREAL;
END_VAR
parent_builder^.Position(value);
Position := parent_builder^.AbsoluteMoveBuilder;
END_METHOD

METHOD PUBLIC Reset : VelocityMoveBuilder
parent_builder^.Reset();
Reset := THIS^;
END_METHOD

METHOD PUBLIC Velocity : VelocityMoveBuilder
VAR_INPUT
	value : LREAL;
END_VAR
parent_builder^.Velocity(value);
Velocity := THIS^;
END_METHOD

END_FUNCTION_BLOCK

// ---- Commands/PointToPoint/MoveVelocityCommand.TcPOU
{attribute 'linkalways'} 
{attribute 'no_explicit_call' := 'This FB is a CLASS and must be accessed using methods or properties'}
{attribute 'enable_dynamic_creation'}
FUNCTION_BLOCK MoveVelocityCommand EXTENDS Mc2MotionCommand
VAR
	fb : Tc2_Mc2.Mc_MoveVelocity;
END_VAR

{attribute 'monitoring' := 'call'}
PROPERTY PUBLIC Active : BOOL
GET // PUBLIC
Active := fb.Active;
END_GET
END_PROPERTY

METHOD PUBLIC CyclicCall
SUPER^.CyclicCall();
fb(Axis := axis_ref);
END_METHOD

(*FB_Init is always available implicitly and it is used primarily for initialization.
The return value is not evaluated. For a specific influence, you can also declare the
methods explicitly and provide additional code there with the standard initialization
code. You can evaluate the return value.*)
METHOD FB_Init : BOOL
VAR_INPUT
	(* TRUE: the retain variables are initialized (reset warm / reset cold)*)
	bInitRetains : BOOL;
	(* TRUE: the instance will be copied to the copy code afterward (online change)*)
	bInCopyCode	: BOOL;
	axis : Axis;
	velocity : LREAL;
	acceleration : LREAL := 0;
	deceleration : LREAL := 0;
	jerk : LREAL := 0;
	buffer_mode	: MotionBufferMode := MotionBufferMode.Aborting;
END_VAR
fb.Velocity := velocity;
fb.Acceleration := acceleration;
fb.Deceleration := deceleration;
fb.Jerk := jerk;
fb.BufferMode := Mc2BufferModeConvertTo(buffer_mode);
END_METHOD

METHOD PROTECTED OnExecuting
VAR_INPUT
	state_control : AsyncCommandStateControl;
END_VAR
fb.Execute := TRUE;

IF fb.InVelocity THEN
	state_control.Next();
	fb.Execute := FALSE;
END_IF

IF fb.CommandAborted THEN
	Abort();
	fb.Execute := FALSE;
END_IF

IF fb.Error THEN
	state_control.Error(fb.ErrorId);
	fb.Execute := FALSE;
END_IF
END_METHOD

END_FUNCTION_BLOCK

// ---- Builders/Motion/Implementation/DefaultAbsoluteMoveBuilder.TcPOU
{attribute 'linkalways'} 
{attribute 'no_explicit_call' := 'This FB is a CLASS and must be accessed using methods or properties'}
{attribute 'enable_dynamic_creation'}
FUNCTION_BLOCK INTERNAL DefaultAbsoluteMoveBuilder IMPLEMENTS AbsoluteMoveBuilder
VAR
	parent_builder : POINTER TO DefaultMotionBuilder;
END_VAR

METHOD PUBLIC Acceleration : AbsoluteMoveBuilder
VAR_INPUT
	value : LREAL;
END_VAR
parent_builder^.Acceleration(value);
Acceleration := THIS^;
END_METHOD

METHOD PUBLIC BufferMode : AbsoluteMoveBuilder
VAR_INPUT
	mode : MotionBufferMode;
END_VAR
parent_builder^.BufferMode(mode);
BufferMode := THIS^;
END_METHOD

METHOD PUBLIC BuildMoveAbsoluteCommand : MotionCommand
VAR_INPUT
	axis : Axis;
END_VAR
VAR
	command_ptr : POINTER TO MoveAbsoluteCommand;
	command : MotionCommand;
END_VAR
command_ptr := __NEW(MoveAbsoluteCommand(
	axis := axis,
	position := parent_builder^.Parameters.position,
	velocity := parent_builder^.Parameters.velocity,
	acceleration := parent_builder^.Parameters.acceleration,
	deceleration := parent_builder^.Parameters.deceleration,
	jerk := parent_builder^.Parameters.jerk,
	buffer_mode := parent_builder^.Parameters.buffer_mode
));
BuildMoveAbsoluteCommand := command_ptr^;
END_METHOD

METHOD PUBLIC Deceleration : AbsoluteMoveBuilder
VAR_INPUT
	value : LREAL;
END_VAR
parent_builder^.Deceleration(value);
Deceleration := THIS^;
END_METHOD

//FB_Init is always available implicitly and it is used primarily for initialization.
//The return value is not evaluated. For a specific influence, you can also declare the
//methods explicitly and provide additional code there with the standard initialization
//code. You can evaluate the return value.
METHOD FB_Init: BOOL
VAR_INPUT
    bInitRetains : BOOL; // TRUE: the retain variables are initialized (reset warm / reset cold)
    bInCopyCode : BOOL;  // TRUE: the instance will be copied to the copy code afterward (online change)
	parent_builder : POINTER TO DefaultMotionBuilder;
END_VAR
THIS^.parent_builder := parent_builder;
END_METHOD

METHOD PUBLIC Jerk : AbsoluteMoveBuilder
VAR_INPUT
	value : LREAL;
END_VAR
parent_builder^.Jerk(value);
Jerk := THIS^;
END_METHOD

METHOD PUBLIC Position : AbsoluteMoveBuilder
VAR_INPUT
	value : LREAL;
END_VAR
parent_builder^.Position(value);
Position := THIS^;
END_METHOD

METHOD PUBLIC Reset : AbsoluteMoveBuilder
parent_builder^.Reset();
Reset := THIS^;
END_METHOD

METHOD PUBLIC Velocity : AbsoluteMoveBuilder
VAR_INPUT
	value : LREAL;
END_VAR
parent_builder^.Velocity(value);
Velocity := THIS^;
END_METHOD

END_FUNCTION_BLOCK

// ---- Commands/PointToPoint/MoveAbsoluteCommand.TcPOU
{attribute 'linkalways'} 
{attribute 'no_explicit_call' := 'This FB is a CLASS and must be accessed using methods or properties'}
{attribute 'enable_dynamic_creation'}
FUNCTION_BLOCK MoveAbsoluteCommand EXTENDS Mc2MotionCommand
VAR
	fb : Tc2_Mc2.Mc_MoveAbsolute;
END_VAR

{attribute 'monitoring' := 'call'}
PROPERTY PUBLIC Active : BOOL
GET // PUBLIC
Active := fb.Active;
END_GET
END_PROPERTY

METHOD PUBLIC CyclicCall
SUPER^.CyclicCall();
fb(Axis := axis_ref);
END_METHOD

(*FB_Init is always available implicitly and it is used primarily for initialization.
The return value is not evaluated. For a specific influence, you can also declare the
methods explicitly and provide additional code there with the standard initialization
code. You can evaluate the return value.*)
METHOD FB_Init : BOOL
VAR_INPUT
	(* TRUE: the retain variables are initialized (reset warm / reset cold)*)
	bInitRetains : BOOL;
	(* TRUE: the instance will be copied to the copy code afterward (online change)*)
	bInCopyCode	: BOOL;
	axis : Axis;
	position : LREAL;
	velocity : LREAL;
	acceleration : LREAL := 0;
	deceleration : LREAL := 0;
	jerk : LREAL := 0;
	buffer_mode	: MotionBufferMode := MotionBufferMode.Aborting;
END_VAR
fb.Position := position;
fb.Velocity := velocity;
fb.Acceleration := acceleration;
fb.Deceleration := deceleration;
fb.Jerk := jerk;
fb.BufferMode := Mc2BufferModeConvertTo(buffer_mode);
END_METHOD

METHOD PROTECTED OnExecuting
VAR_INPUT
	state_control : AsyncCommandStateControl;
END_VAR
fb.Execute := TRUE;

IF fb.Done THEN
	fb.Execute := FALSE;
	state_control.Next();
END_IF

IF fb.CommandAborted THEN
	fb.Execute := FALSE;
	Abort();
END_IF

IF fb.Error THEN
	fb.Execute := FALSE;
	state_control.Error(fb.ErrorId);
END_IF
END_METHOD

END_FUNCTION_BLOCK

// ---- Builders/Motion/Implementation/DefaultRelativeMoveBuilder.TcPOU
{attribute 'linkalways'} 
{attribute 'no_explicit_call' := 'This FB is a CLASS and must be accessed using methods or properties'}
{attribute 'enable_dynamic_creation'}
FUNCTION_BLOCK INTERNAL DefaultRelativeMoveBuilder IMPLEMENTS RelativeMoveBuilder
VAR
	parent_builder : POINTER TO DefaultMotionBuilder;
END_VAR

METHOD PUBLIC Acceleration : RelativeMoveBuilder
VAR_INPUT
	value : LREAL;
END_VAR
parent_builder^.Acceleration(value);
Acceleration := THIS^;
END_METHOD

METHOD PUBLIC BufferMode : RelativeMoveBuilder
VAR_INPUT
	mode : MotionBufferMode;
END_VAR
parent_builder^.BufferMode(mode);
BufferMode := THIS^;
END_METHOD

METHOD PUBLIC BuildMoveAdditiveCommand : MotionCommand
VAR_INPUT
	axis : Axis;
END_VAR
VAR
	command_ptr : POINTER TO MoveAdditiveCommand;
	command : MotionCommand;
END_VAR
command_ptr := __NEW(MoveAdditiveCommand(
	axis := axis,
	distance := parent_builder^.Parameters.distance,
	velocity := parent_builder^.Parameters.velocity,
	acceleration := parent_builder^.Parameters.acceleration,
	deceleration := parent_builder^.Parameters.deceleration,
	jerk := parent_builder^.Parameters.jerk,
	buffer_mode := parent_builder^.Parameters.buffer_mode
));
BuildMoveAdditiveCommand := command_ptr^;
END_METHOD

METHOD PUBLIC BuildMoveRelativeCommand : MotionCommand
VAR_INPUT
	axis : Axis;
END_VAR
VAR
	command_ptr : POINTER TO MoveRelativeCommand;
	command : MotionCommand;
END_VAR
command_ptr := __NEW(MoveRelativeCommand(
	axis := axis,
	distance := parent_builder^.Parameters.distance,
	velocity := parent_builder^.Parameters.velocity,
	acceleration := parent_builder^.Parameters.acceleration,
	deceleration := parent_builder^.Parameters.deceleration,
	jerk := parent_builder^.Parameters.jerk,
	buffer_mode := parent_builder^.Parameters.buffer_mode
));
BuildMoveRelativeCommand := command_ptr^;
END_METHOD

METHOD PUBLIC Deceleration : RelativeMoveBuilder
VAR_INPUT
	value : LREAL;
END_VAR
parent_builder^.Deceleration(value);
Deceleration := THIS^;
END_METHOD

METHOD PUBLIC Distance : RelativeMoveBuilder
VAR_INPUT
	value : LREAL;
END_VAR
parent_builder^.Distance(value);
Distance := THIS^;
END_METHOD

//FB_Init is always available implicitly and it is used primarily for initialization.
//The return value is not evaluated. For a specific influence, you can also declare the
//methods explicitly and provide additional code there with the standard initialization
//code. You can evaluate the return value.
METHOD FB_Init: BOOL
VAR_INPUT
    bInitRetains : BOOL; // TRUE: the retain variables are initialized (reset warm / reset cold)
    bInCopyCode : BOOL;  // TRUE: the instance will be copied to the copy code afterward (online change)
	parent_builder : POINTER TO DefaultMotionBuilder;
END_VAR
THIS^.parent_builder := parent_builder;
END_METHOD

METHOD PUBLIC Jerk : RelativeMoveBuilder
VAR_INPUT
	value : LREAL;
END_VAR
parent_builder^.Jerk(value);
Jerk := THIS^;
END_METHOD

METHOD PUBLIC Reset : RelativeMoveBuilder
parent_builder^.Reset();
Reset := THIS^;
END_METHOD

METHOD PUBLIC Velocity : RelativeMoveBuilder
VAR_INPUT
	value : LREAL;
END_VAR
parent_builder^.Velocity(value);
Velocity := THIS^;
END_METHOD

END_FUNCTION_BLOCK

// ---- Commands/PointToPoint/MoveAdditiveCommand.TcPOU
{attribute 'linkalways'} 
{attribute 'no_explicit_call' := 'This FB is a CLASS and must be accessed using methods or properties'}
{attribute 'enable_dynamic_creation'}
FUNCTION_BLOCK MoveAdditiveCommand EXTENDS Mc2MotionCommand
VAR
	fb : Tc2_Mc2.Mc_MoveAdditive;
END_VAR

{attribute 'monitoring' := 'call'}
PROPERTY PUBLIC Active : BOOL
GET // PUBLIC
Active := fb.Active;
END_GET
END_PROPERTY

METHOD PUBLIC CyclicCall
SUPER^.CyclicCall();
fb(Axis := axis_ref);
END_METHOD

(*FB_Init is always available implicitly and it is used primarily for initialization.
The return value is not evaluated. For a specific influence, you can also declare the
methods explicitly and provide additional code there with the standard initialization
code. You can evaluate the return value.*)
METHOD FB_Init : BOOL
VAR_INPUT
	(* TRUE: the retain variables are initialized (reset warm / reset cold)*)
	bInitRetains : BOOL;
	(* TRUE: the instance will be copied to the copy code afterward (online change)*)
	bInCopyCode	: BOOL;
	axis : Axis;
	distance : LREAL;
	velocity : LREAL;
	acceleration : LREAL := 0;
	deceleration : LREAL := 0;
	jerk : LREAL := 0;
	buffer_mode	: MotionBufferMode := MotionBufferMode.Aborting;
END_VAR
fb.Distance := distance;
fb.Velocity := velocity;
fb.Acceleration := acceleration;
fb.Deceleration := deceleration;
fb.Jerk := jerk;
fb.BufferMode := Mc2BufferModeConvertTo(buffer_mode);
END_METHOD

METHOD PROTECTED OnExecuting
VAR_INPUT
	state_control : AsyncCommandStateControl;
END_VAR
fb.Execute := TRUE;

IF fb.Done THEN
	state_control.Next();
	fb.Execute := FALSE;
END_IF

IF fb.CommandAborted THEN
	Abort();
	fb.Execute := FALSE;
END_IF

IF fb.Error THEN
	state_control.Error(fb.ErrorId);
	fb.Execute := FALSE;
END_IF
END_METHOD

END_FUNCTION_BLOCK

// ---- Commands/PointToPoint/MoveRelativeCommand.TcPOU
{attribute 'linkalways'} 
{attribute 'no_explicit_call' := 'This FB is a CLASS and must be accessed using methods or properties'}
{attribute 'enable_dynamic_creation'}
FUNCTION_BLOCK MoveRelativeCommand EXTENDS Mc2MotionCommand
VAR
	fb : Tc2_Mc2.Mc_MoveRelative;
END_VAR

{attribute 'monitoring' := 'call'}
PROPERTY PUBLIC Active : BOOL
GET // PUBLIC
Active := fb.Active;
END_GET
END_PROPERTY

METHOD PUBLIC CyclicCall
SUPER^.CyclicCall();
fb(Axis := axis_ref);
END_METHOD

(*FB_Init is always available implicitly and it is used primarily for initialization.
The return value is not evaluated. For a specific influence, you can also declare the
methods explicitly and provide additional code there with the standard initialization
code. You can evaluate the return value.*)
METHOD FB_Init : BOOL
VAR_INPUT
	(* TRUE: the retain variables are initialized (reset warm / reset cold)*)
	bInitRetains : BOOL;
	(* TRUE: the instance will be copied to the copy code afterward (online change)*)
	bInCopyCode	: BOOL;
	axis : Axis;
	distance : LREAL;
	velocity : LREAL;
	acceleration : LREAL := 0;
	deceleration : LREAL := 0;
	jerk : LREAL := 0;
	buffer_mode	: MotionBufferMode := MotionBufferMode.Aborting;
END_VAR
fb.Distance := distance;
fb.Velocity := velocity;
fb.Acceleration := acceleration;
fb.Deceleration := deceleration;
fb.Jerk := jerk;
fb.BufferMode := Mc2BufferModeConvertTo(buffer_mode);
END_METHOD

METHOD PROTECTED OnExecuting
VAR_INPUT
	state_control : AsyncCommandStateControl;
END_VAR
fb.Execute := TRUE;

IF fb.Done THEN
	state_control.Next();
	fb.Execute := FALSE;
END_IF

IF fb.CommandAborted THEN
	Abort();
	fb.Execute := FALSE;
END_IF

IF fb.Error THEN
	state_control.Error(fb.ErrorId);
	fb.Execute := FALSE;
END_IF
END_METHOD

END_FUNCTION_BLOCK

// ---- Commands/Stops/StopCommand.TcPOU
{attribute 'linkalways'} 
{attribute 'no_explicit_call' := 'This FB is a CLASS and must be accessed using methods or properties'}
{attribute 'enable_dynamic_creation'}
FUNCTION_BLOCK StopCommand EXTENDS Mc2MotionCommand
VAR
	fb : Tc2_Mc2.Mc_Stop;
END_VAR

{attribute 'monitoring' := 'call'}
PROPERTY PUBLIC Active : BOOL
GET // PUBLIC
Active := fb.Active;
END_GET
END_PROPERTY

METHOD PUBLIC CyclicCall
SUPER^.CyclicCall();
fb(Axis := axis_ref);
END_METHOD

(*FB_Init is always available implicitly and it is used primarily for initialization.
The return value is not evaluated. For a specific influence, you can also declare the
methods explicitly and provide additional code there with the standard initialization
code. You can evaluate the return value.*)
METHOD FB_Init : BOOL
VAR_INPUT
	(* TRUE: the retain variables are initialized (reset warm / reset cold)*)
	bInitRetains : BOOL;
	(* TRUE: the instance will be copied to the copy code afterward (online change)*)
	bInCopyCode	: BOOL;
	axis : Axis;
	deceleration : LREAL := 0;
	jerk : LREAL := 0;
END_VAR
fb.Deceleration := deceleration;
fb.Jerk := jerk;
END_METHOD

METHOD PROTECTED OnExecuting
VAR_INPUT
	state_control : AsyncCommandStateControl;
END_VAR
fb.Execute := TRUE;

IF fb.Done THEN
	state_control.Next();
	fb.Execute := FALSE;
END_IF

IF fb.CommandAborted THEN
	Abort();
	fb.Execute := FALSE;
END_IF

IF fb.Error THEN
	state_control.Error(fb.ErrorId);
	fb.Execute := FALSE;
END_IF
END_METHOD

END_FUNCTION_BLOCK

// ---- Commands/Coupling/GearInCommand.TcPOU
{attribute 'linkalways'} 
{attribute 'no_explicit_call' := 'This FB is a CLASS and must be accessed using methods or properties'}
{attribute 'enable_dynamic_creation'}
FUNCTION_BLOCK GearInCommand EXTENDS NoopAsyncCommand IMPLEMENTS AsyncCommand
VAR
	master_axis_ref : REFERENCE TO Tc2_Mc2.Axis_Ref;
	slave_axis_ref : REFERENCE TO Tc2_Mc2.Axis_Ref;
	fb : Tc2_Mc2.Mc_GearIn;
END_VAR

METHOD PUBLIC CyclicCall
SUPER^.CyclicCall();
fb(Master := master_axis_ref, Slave := slave_axis_ref);
END_METHOD

(*FB_Init is always available implicitly and it is used primarily for initialization.
The return value is not evaluated. For a specific influence, you can also declare the
methods explicitly and provide additional code there with the standard initialization
code. You can evaluate the return value.*)
METHOD FB_Init : BOOL
VAR_INPUT
	(* TRUE: the retain variables are initialized (reset warm / reset cold)*)
	bInitRetains : BOOL;
	(* TRUE: the instance will be copied to the copy code afterward (online change)*)
	bInCopyCode	: BOOL;
	master_axis : Axis;
	slave_axis : Axis;
	numerator : LREAL;
	denominator : UINT := 1;
END_VAR
master_axis_ref REF= master_axis.AxisRef;
slave_axis_ref REF= slave_axis.AxisRef;
fb.RatioNumerator := numerator;
fb.RatioDenominator := denominator;
END_METHOD

METHOD PROTECTED OnExecuting
VAR_INPUT
	state_control : AsyncCommandStateControl;
END_VAR
fb.Execute := TRUE;

IF fb.InGear THEN
	state_control.Next();
	fb.Execute := FALSE;
END_IF

IF fb.CommandAborted THEN
	Abort();
	fb.Execute := FALSE;
END_IF

IF fb.Error THEN
	state_control.Error(fb.ErrorId);
	fb.Execute := FALSE;
END_IF
END_METHOD

END_FUNCTION_BLOCK

// ---- Commands/SoE/ResetSoeDriveCommand.TcPOU
{attribute 'linkalways'} 
{attribute 'no_explicit_call' := 'This FB is a CLASS and must be accessed using methods or properties'}
{attribute 'enable_dynamic_creation'}
FUNCTION_BLOCK PUBLIC ResetSoeDriveCommand EXTENDS Mc2MotionCommand IMPLEMENTS AsyncCommand
VAR
	fb : Tc2_Mc2_Drive.Fb_SoeReset;
END_VAR

METHOD PUBLIC CyclicCall
SUPER^.CyclicCall();
fb(Axis := axis_ref, Timeout := T#5S);
END_METHOD

METHOD PROTECTED OnExecuting
VAR_INPUT
	state_control : AsyncCommandStateControl;
END_VAR
fb.Execute := TRUE;

if NOT fb.Busy then
	if fb.Error then
		state_control.Error(fb.AdsErrId);
	ELSE
		state_control.Next();
	END_IF
	fb.Execute := FALSE;
END_IF
END_METHOD

END_FUNCTION_BLOCK

// ---- Commands/PointToPoint/MoveContinuousAbsoluteCommand.TcPOU
{attribute 'linkalways'} 
{attribute 'no_explicit_call' := 'This FB is a CLASS and must be accessed using methods or properties'}
{attribute 'enable_dynamic_creation'}
FUNCTION_BLOCK MoveContinuousAbsoluteCommand EXTENDS Mc2MotionCommand
VAR
	fb : Tc2_Mc2.Mc_MoveContinuousAbsolute;
END_VAR

{attribute 'monitoring' := 'call'}
PROPERTY PUBLIC Active : BOOL
GET // PUBLIC
Active := fb.Active;
END_GET
END_PROPERTY

METHOD PUBLIC CyclicCall
SUPER^.CyclicCall();
fb(Axis := axis_ref);
END_METHOD

(*FB_Init is always available implicitly and it is used primarily for initialization.
The return value is not evaluated. For a specific influence, you can also declare the
methods explicitly and provide additional code there with the standard initialization
code. You can evaluate the return value.*)
METHOD FB_Init : BOOL
VAR_INPUT
	(* TRUE: the retain variables are initialized (reset warm / reset cold)*)
	bInitRetains : BOOL;
	(* TRUE: the instance will be copied to the copy code afterward (online change)*)
	bInCopyCode	: BOOL;
	axis : Axis;
	position : LREAL;
	velocity : LREAL;
	acceleration : LREAL := 0;
	deceleration : LREAL := 0;
	jerk : LREAL := 0;
	buffer_mode	: MotionBufferMode := MotionBufferMode.Aborting;
END_VAR
fb.Position := position;
fb.Velocity := velocity;
fb.Acceleration := acceleration;
fb.Deceleration := deceleration;
fb.Jerk := jerk;
fb.BufferMode := Mc2BufferModeConvertTo(buffer_mode);
END_METHOD

METHOD PROTECTED OnExecuting
VAR_INPUT
	state_control : AsyncCommandStateControl;
END_VAR
fb.Execute := TRUE;

IF fb.InEndVelocity THEN
	state_control.Next();
	fb.Execute := FALSE;
END_IF

IF fb.CommandAborted THEN
	Abort();
	fb.Execute := FALSE;
END_IF

IF fb.Error THEN
	state_control.Error(fb.ErrorId);
	fb.Execute := FALSE;
END_IF
END_METHOD

END_FUNCTION_BLOCK

// ---- Commands/PointToPoint/MoveContinuousRelativeCommand.TcPOU
{attribute 'linkalways'} 
{attribute 'no_explicit_call' := 'This FB is a CLASS and must be accessed using methods or properties'}
{attribute 'enable_dynamic_creation'}
FUNCTION_BLOCK MoveContinuousRelativeCommand EXTENDS Mc2MotionCommand
VAR
	fb : Tc2_Mc2.Mc_MoveContinuousRelative;
END_VAR

{attribute 'monitoring' := 'call'}
PROPERTY PUBLIC Active : BOOL
GET // PUBLIC
Active := fb.Active;
END_GET
END_PROPERTY

METHOD PUBLIC CyclicCall
SUPER^.CyclicCall();
fb(Axis := axis_ref);
END_METHOD

(*FB_Init is always available implicitly and it is used primarily for initialization.
The return value is not evaluated. For a specific influence, you can also declare the
methods explicitly and provide additional code there with the standard initialization
code. You can evaluate the return value.*)
METHOD FB_Init : BOOL
VAR_INPUT
	(* TRUE: the retain variables are initialized (reset warm / reset cold)*)
	bInitRetains : BOOL;
	(* TRUE: the instance will be copied to the copy code afterward (online change)*)
	bInCopyCode	: BOOL;
	axis : Axis;
	distance : LREAL;
	velocity : LREAL;
	acceleration : LREAL := 0;
	deceleration : LREAL := 0;
	jerk : LREAL := 0;
	buffer_mode	: MotionBufferMode := MotionBufferMode.Aborting;
END_VAR
fb.Distance := distance;
fb.Velocity := velocity;
fb.Acceleration := acceleration;
fb.Deceleration := deceleration;
fb.Jerk := jerk;
fb.BufferMode := Mc2BufferModeConvertTo(buffer_mode);
END_METHOD

METHOD PROTECTED OnExecuting
VAR_INPUT
	state_control : AsyncCommandStateControl;
END_VAR
fb.Execute := TRUE;

IF fb.InEndVelocity THEN
	state_control.Next();
	fb.Execute := FALSE;
END_IF

IF fb.CommandAborted THEN
	Abort();
	fb.Execute := FALSE;
END_IF

IF fb.Error THEN
	state_control.Error(fb.ErrorId);
	fb.Execute := FALSE;
END_IF
END_METHOD

END_FUNCTION_BLOCK

// ---- Commands/PointToPoint/MoveModuloCommand.TcPOU
{attribute 'linkalways'} 
{attribute 'no_explicit_call' := 'This FB is a CLASS and must be accessed using methods or properties'}
{attribute 'enable_dynamic_creation'}
FUNCTION_BLOCK MoveModuloCommand EXTENDS Mc2MotionCommand
VAR
	fb : Tc2_Mc2.Mc_MoveModulo;
END_VAR

{attribute 'monitoring' := 'call'}
PROPERTY PUBLIC Active : BOOL
GET // PUBLIC
Active := fb.Active;
END_GET
END_PROPERTY

METHOD PUBLIC CyclicCall
SUPER^.CyclicCall();
fb(Axis := axis_ref);
END_METHOD

(*FB_Init is always available implicitly and it is used primarily for initialization.
The return value is not evaluated. For a specific influence, you can also declare the
methods explicitly and provide additional code there with the standard initialization
code. You can evaluate the return value.*)
METHOD FB_Init : BOOL
VAR_INPUT
	(* TRUE: the retain variables are initialized (reset warm / reset cold)*)
	bInitRetains : BOOL;
	(* TRUE: the instance will be copied to the copy code afterward (online change)*)
	bInCopyCode	: BOOL;
	axis : Axis;
	position : LREAL;
	direction : MotionDirection;
	velocity : LREAL;
	acceleration : LREAL := 0;
	deceleration : LREAL := 0;
	jerk : LREAL := 0;
	buffer_mode	: MotionBufferMode := MotionBufferMode.Aborting;
END_VAR
fb.Position := position;
fb.Direction := Mc2DirectionConvertTo(direction);
fb.Velocity := velocity;
fb.Acceleration := acceleration;
fb.Deceleration := deceleration;
fb.Jerk := jerk;
fb.BufferMode := Mc2BufferModeConvertTo(buffer_mode);
END_METHOD

METHOD PROTECTED OnExecuting
VAR_INPUT
	state_control : AsyncCommandStateControl;
END_VAR
fb.Execute := TRUE;

IF fb.Done THEN
	state_control.Next();
	fb.Execute := FALSE;
END_IF

IF fb.CommandAborted THEN
	Abort();
	fb.Execute := FALSE;
END_IF

IF fb.Error THEN
	state_control.Error(fb.ErrorId);
	fb.Execute := FALSE;
END_IF
END_METHOD

END_FUNCTION_BLOCK

// ---- Functions/Mc2DirectionConvertTo.TcPOU
FUNCTION INTERNAL Mc2DirectionConvertTo : Tc2_Mc2.Mc_Direction
VAR_INPUT
	direction : MotionDirection;
END_VAR

CASE direction OF
	MotionDirection.Positive: Mc2DirectionConvertTo := Tc2_Mc2.Mc_Direction.Mc_Positive_Direction;
	MotionDirection.ShortestWay: Mc2DirectionConvertTo := Tc2_Mc2.Mc_Direction.Mc_Shortest_Way;
	MotionDirection.Negative: Mc2DirectionConvertTo := Tc2_Mc2.Mc_Direction.Mc_Negative_Direction;
	MotionDirection.Current: Mc2DirectionConvertTo := Tc2_Mc2.Mc_Direction.Mc_Current_Direction;
	MotionDirection.Undefined: Mc2DirectionConvertTo := Tc2_Mc2.Mc_Direction.Mc_Undefined_Direction;
END_CASE

END_FUNCTION

// ---- Functions/Mc2BufferModeConvertFrom.TcPOU
FUNCTION INTERNAL Mc2BufferModeConvertFrom : MotionBufferMode
VAR_INPUT
	buffer_mode : Tc2_Mc2.Mc_BufferMode;
END_VAR

CASE buffer_mode OF
	Tc2_Mc2.Mc_BufferMode.Mc_Aborting: Mc2BufferModeConvertFrom := MotionBufferMode.Aborting;
    Tc2_Mc2.Mc_BufferMode.Mc_Buffered: Mc2BufferModeConvertFrom := MotionBufferMode.Buffered;
    Tc2_Mc2.Mc_BufferMode.Mc_BlendingLow: Mc2BufferModeConvertFrom := MotionBufferMode.BlendingLow;
   	Tc2_Mc2.Mc_BufferMode.Mc_BlendingPrevious: Mc2BufferModeConvertFrom := MotionBufferMode.BlendingPrevious;
    Tc2_Mc2.Mc_BufferMode.Mc_BlendingNext: Mc2BufferModeConvertFrom := MotionBufferMode.BlendingNext;
    Tc2_Mc2.Mc_BufferMode.Mc_BlendingHigh: Mc2BufferModeConvertFrom := MotionBufferMode.BlendingHigh;
END_CASE

END_FUNCTION

// ---- Functions/Mc2DirectionConvertFrom.TcPOU
FUNCTION INTERNAL Mc2DirectionConvertFrom : MotionDirection
VAR_INPUT
	direction : Tc2_Mc2.Mc_Direction;
END_VAR

CASE direction OF
	Tc2_Mc2.Mc_Direction.Mc_Positive_Direction: Mc2DirectionConvertFrom := MotionDirection.Positive;
	Tc2_Mc2.Mc_Direction.Mc_Shortest_Way: Mc2DirectionConvertFrom := MotionDirection.ShortestWay;
	Tc2_Mc2.Mc_Direction.Mc_Negative_Direction: Mc2DirectionConvertFrom := MotionDirection.Negative;
	Tc2_Mc2.Mc_Direction.Mc_Current_Direction: Mc2DirectionConvertFrom := MotionDirection.Current;
	Tc2_Mc2.Mc_Direction.Mc_Undefined_Direction: Mc2DirectionConvertFrom := MotionDirection.Undefined;
END_CASE

END_FUNCTION

// ---- Axis/Mc2Axis.TcPOU
{attribute 'linkalways'} 
{attribute 'no_explicit_call' := 'This FB is a CLASS and must be accessed using methods or properties'}
{attribute 'enable_dynamic_creation'}
FUNCTION_BLOCK Mc2Axis IMPLEMENTS Axis
VAR
	axis_ref : Tc2_Mc2.Axis_Ref;
	power_fb : Tc2_Mc2.Mc_Power;
	halt_fb : Tc2_Mc2.Mc_Halt;
	stop_fb : Tc2_Mc2.Mc_Stop;
	
	reset_command : ResetCommand(axis := THIS^);
	reset_drive_command : ResetSoeDriveCommand(axis := THIS^);
END_VAR

{attribute 'monitoring' := 'call'}
PROPERTY PUBLIC ActualAcceleration : LREAL
GET // PUBLIC
ActualAcceleration := axis_ref.NcToPlc.ActAcc;
END_GET
END_PROPERTY

{attribute 'monitoring' := 'call'}
PROPERTY PUBLIC ActualPosition : LREAL
GET // PUBLIC
ActualPosition := axis_ref.NcToPlc.ActPos;
END_GET
END_PROPERTY

{attribute 'monitoring' := 'call'}
PROPERTY PUBLIC ActualVelocity : LREAL
GET // PUBLIC
ActualVelocity := axis_ref.NcToPlc.ActVelo;
END_GET
END_PROPERTY

PROPERTY PUBLIC AxisRef : REFERENCE TO Tc2_Mc2.Axis_Ref
GET // PUBLIC
AxisRef REF= THIS^.axis_ref;
END_GET
END_PROPERTY

METHOD PUBLIC CyclicCall
power_fb(Axis := axis_ref);
reset_command.CyclicCall();
reset_drive_command.CyclicCall();
halt_fb(Axis := axis_ref);
stop_fb(Axis := axis_ref);
axis_ref.ReadStatus();
END_METHOD

METHOD PUBLIC Disable
power_fb.Enable := FALSE;
power_fb.Enable_Positive := FALSE;
power_fb.Enable_Negative := FALSE;
END_METHOD

METHOD PUBLIC DisableNegative
power_fb.Enable_Negative := FALSE;
END_METHOD

METHOD PUBLIC DisablePositive
power_fb.Enable_Positive := FALSE;
END_METHOD

METHOD PUBLIC Enable
power_fb.Enable := TRUE;
END_METHOD

METHOD PUBLIC EnableNegative
power_fb.Enable_Negative := TRUE;
END_METHOD

METHOD PUBLIC EnablePositive
power_fb.Enable_Positive := TRUE;
END_METHOD

{attribute 'monitoring' := 'call'}
PROPERTY PUBLIC ErrorId : UDINT
GET // PUBLIC
ErrorId := axis_ref.Status.ErrorId;
END_GET
END_PROPERTY

{attribute 'monitoring' := 'call'}
PROPERTY PUBLIC HasBeenStopped : BOOL
GET // PUBLIC
HasBeenStopped := axis_ref.Status.HasBeenStopped;
END_GET
END_PROPERTY

{attribute 'monitoring' := 'call'}
PROPERTY PUBLIC HasJob : BOOL
GET // PUBLIC
HasJob := axis_ref.Status.HasJob;
END_GET
END_PROPERTY

{attribute 'monitoring' := 'call'}
PROPERTY PUBLIC IsAccelerating : BOOL
GET // PUBLIC
IsAccelerating := axis_ref.Status.Accelerating;
END_GET
END_PROPERTY

{attribute 'monitoring' := 'call'}
PROPERTY PUBLIC IsBusyHoming : BOOL
GET // PUBLIC
IsBusyHoming := axis_ref.Status.HomingBusy;
END_GET
END_PROPERTY

{attribute 'monitoring' := 'call'}
PROPERTY PUBLIC IsCamDataQueued : BOOL
GET // PUBLIC
IsCamDataQueued := axis_ref.Status.CamDataQueued;
END_GET
END_PROPERTY

{attribute 'monitoring' := 'call'}
PROPERTY PUBLIC IsCamScalingPending : BOOL
GET // PUBLIC
IsCamScalingPending := axis_ref.Status.CamScalingPending;
END_GET
END_PROPERTY

{attribute 'monitoring' := 'call'}
PROPERTY PUBLIC IsCamTableQueued : BOOL
GET // PUBLIC
IsCamTableQueued := axis_ref.Status.CamTableQueued;
END_GET
END_PROPERTY

{attribute 'monitoring' := 'call'}
 PROPERTY PUBLIC IsCommandBuffered : BOOL
GET // PUBLIC
IsCommandBuffered := axis_ref.Status.CmdBuffered;
END_GET
END_PROPERTY

{attribute 'monitoring' := 'call'}
PROPERTY PUBLIC IsCompensating : BOOL
GET // PUBLIC
IsCompensating := axis_ref.Status.Compensating;
END_GET
END_PROPERTY

{attribute 'monitoring' := 'call'}
PROPERTY PUBLIC IsConstantVelocity : BOOL
GET // PUBLIC
IsConstantVelocity := axis_ref.Status.ConstantVelocity;
END_GET
END_PROPERTY

{attribute 'monitoring' := 'call'}
PROPERTY PUBLIC IsContinuousMotion : BOOL
GET // PUBLIC
IsContinuousMotion := axis_ref.Status.ContinuousMotion;
END_GET
END_PROPERTY

{attribute 'monitoring' := 'call'}
PROPERTY PUBLIC IsControlLoopClosed : BOOL
GET // PUBLIC
IsControlLoopClosed := axis_ref.Status.ControlLoopClosed;
END_GET
END_PROPERTY

{attribute 'monitoring' := 'call'}
PROPERTY PUBLIC IsCoupled : BOOL
GET // PUBLIC
IsCoupled := axis_ref.Status.Coupled;
END_GET
END_PROPERTY

{attribute 'monitoring' := 'call'}
PROPERTY PUBLIC IsDecelerating : BOOL
GET // PUBLIC
IsDecelerating := axis_ref.Status.Decelerating;
END_GET
END_PROPERTY

{attribute 'monitoring' := 'call'}
PROPERTY PUBLIC IsDisabled : BOOL
GET // PUBLIC
IsDisabled := axis_ref.Status.Disabled;
END_GET
END_PROPERTY

{attribute 'monitoring' := 'call'}
PROPERTY PUBLIC IsDiscreteMotion : BOOL
GET // PUBLIC
END_GET
END_PROPERTY

{attribute 'monitoring' := 'call'}
PROPERTY PUBLIC IsDriveDeviceErrored : BOOL
GET // PUBLIC
IsDriveDeviceErrored := axis_ref.Status.Error;
END_GET
END_PROPERTY

{attribute 'monitoring' := 'call'}
PROPERTY PUBLIC IsErrored : BOOL
GET // PUBLIC
IsErrored := axis_ref.Status.Error;
END_GET
END_PROPERTY

{attribute 'monitoring' := 'call'}
PROPERTY PUBLIC IsErrorStop : BOOL
GET // PUBLIC
IsErrorStop := axis_ref.Status.ErrorStop;
END_GET
END_PROPERTY

{attribute 'monitoring' := 'call'}
PROPERTY PUBLIC IsExternalLatchValid : BOOL
GET // PUBLIC
IsExternalLatchValid := axis_ref.Status.ExternalLatchValid;
END_GET
END_PROPERTY

{attribute 'monitoring' := 'call'}
PROPERTY PUBLIC IsExtSetPointGenEnabled : BOOL
GET // PUBLIC
IsExtSetPointGenEnabled := axis_ref.Status.ExtSetPointGenEnabled;
END_GET
END_PROPERTY

{attribute 'monitoring' := 'call'}
PROPERTY PUBLIC IsHomed : BOOL
GET // PUBLIC
IsHomed := axis_ref.Status.Homed;
END_GET
END_PROPERTY

{attribute 'monitoring' := 'call'}
PROPERTY PUBLIC IsHoming : BOOL
GET // PUBLIC
IsHoming := axis_ref.Status.Homing;
END_GET
END_PROPERTY

{attribute 'monitoring' := 'call'}
PROPERTY PUBLIC IsInPositionArea : BOOL
GET // PUBLIC
IsInPositionArea := axis_ref.Status.InPositionArea;
END_GET
END_PROPERTY

{attribute 'monitoring' := 'call'}
PROPERTY PUBLIC IsInTargetPosition : BOOL
GET // PUBLIC
IsInTargetPosition := axis_ref.Status.InTargetPosition;
END_GET
END_PROPERTY

{attribute 'monitoring' := 'call'}
PROPERTY PUBLIC IsIoDataInvalid : BOOL
GET // PUBLIC
IsIoDataInvalid := axis_ref.Status.IoDataInvalid;
END_GET
END_PROPERTY

{attribute 'monitoring' := 'call'}
PROPERTY PUBLIC IsMotionCommandsLocked : BOOL
GET // PUBLIC
IsMotionCommandsLocked := axis_ref.Status.MotionCommandsLocked;
END_GET
END_PROPERTY

{attribute 'monitoring' := 'call'}
PROPERTY PUBLIC IsMoving : BOOL
GET // PUBLIC
IsMoving := axis_ref.Status.Moving;
END_GET
END_PROPERTY

{attribute 'monitoring' := 'call'}
PROPERTY PUBLIC IsNegativeDirection : BOOL
GET // PUBLIC
IsNegativeDirection := axis_ref.Status.NegativeDirection;
END_GET
END_PROPERTY

{attribute 'monitoring' := 'call'}
PROPERTY PUBLIC IsNewTargetPosition : BOOL
GET // PUBLIC
IsNewTargetPosition := axis_ref.Status.NewTargetPosition;
END_GET
END_PROPERTY

{attribute 'monitoring' := 'call'}
PROPERTY PUBLIC IsNotMoving : BOOL
GET // PUBLIC
IsNotMoving := axis_ref.Status.NotMoving;
END_GET
END_PROPERTY

{attribute 'monitoring' := 'call'}
PROPERTY PUBLIC IsOperational : BOOL
GET // PUBLIC
IsOperational := axis_ref.Status.Operational;
END_GET
END_PROPERTY

{attribute 'monitoring' := 'call'}
PROPERTY PUBLIC IsPointToPointMode : BOOL
GET // PUBLIC
IsPointToPointMode := axis_ref.Status.PTPmode;
END_GET
END_PROPERTY

{attribute 'monitoring' := 'call'}
PROPERTY PUBLIC IsPositiveDirection : BOOL
GET // PUBLIC
IsPositiveDirection := axis_ref.Status.PositiveDirection;
END_GET
END_PROPERTY

{attribute 'monitoring' := 'call'}
PROPERTY PUBLIC IsProtected : BOOL
GET // PUBLIC
IsProtected := axis_ref.Status.ProtectedMode;
END_GET
END_PROPERTY

{attribute 'monitoring' := 'call'}
PROPERTY PUBLIC IsSoftLimitMaxExceeded : BOOL
GET // PUBLIC
IsSoftLimitMaxExceeded := axis_ref.Status.SoftLimitMaxExceeded;
END_GET
END_PROPERTY

{attribute 'monitoring' := 'call'}
PROPERTY PUBLIC IsSoftLimitMinExceeded : BOOL
GET // PUBLIC
IsSoftLimitMinExceeded := axis_ref.Status.SoftLimitMinExceeded;
END_GET
END_PROPERTY

{attribute 'monitoring' := 'call'}
PROPERTY PUBLIC IsStandstill : BOOL
GET // PUBLIC
IsStandstill := axis_ref.Status.StandStill;
END_GET
END_PROPERTY

{attribute 'monitoring' := 'call'}
PROPERTY PUBLIC IsStopping : BOOL
GET // PUBLIC
IsStopping := axis_ref.Status.Stopping;
END_GET
END_PROPERTY

{attribute 'monitoring' := 'call'}
PROPERTY PUBLIC IsSynchronisedMotion : BOOL
GET // PUBLIC
IsSynchronisedMotion := axis_ref.Status.SynchronizedMotion;
END_GET
END_PROPERTY

{attribute 'monitoring' := 'call'}
PROPERTY PUBLIC MotionState : AxisMotionState
GET // PUBLIC
CASE axis_ref.Status.MotionState OF
	Tc2_Mc2.Mc_AxisState_Disabled: MotionState := AxisMotionState.Disabled;
	Tc2_Mc2.Mc_AxisState_Standstill: MotionState := AxisMotionState.Standstill;
	Tc2_Mc2.Mc_AxisState_ErrorStop: MotionState := AxisMotionState.ErrorStop;
	Tc2_Mc2.Mc_AxisState_Stopping: MotionState := AxisMotionState.Stopping;
	Tc2_Mc2.Mc_AxisState_Homing: MotionState := AxisMotionState.Homing;
	Tc2_Mc2.Mc_AxisState_DiscreteMotion: MotionState := AxisMotionState.DiscreteMotion;
	Tc2_Mc2.Mc_AxisState_ContinousMotion: MotionState := AxisMotionState.ContinuousMotion;
	Tc2_Mc2.Mc_AxisState_SynchronizedMotion: MotionState := AxisMotionState.SynchronisedMotion;
ELSE
	MotionState := AxisMotionState.Undefined;
END_CASE
END_GET
END_PROPERTY

PROPERTY PUBLIC OpMode : Tc2_Mc2.St_AxisOpModes
GET // PUBLIC
OpMode := axis_ref.Status.OpMode;
END_GET
END_PROPERTY

PROPERTY PUBLIC Override : LREAL
GET // PUBLIC
Override := power_fb.Override;
END_GET
SET // PUBLIC
power_fb.Override := Override;
END_SET
END_PROPERTY

METHOD PUBLIC Reset : AsyncCommand
reset_command.Execute();
Reset := reset_command;
END_METHOD

METHOD PUBLIC ResetDrive : AsyncCommand
reset_drive_command.Execute();
ResetDrive := reset_drive_command;
END_METHOD

{warning 'Add method implementation '}
METHOD PUBLIC SetPosition : AsyncCommand
VAR_INPUT
	position : LREAL;
END_VAR
END_METHOD

{attribute 'monitoring' := 'call'}
PROPERTY PUBLIC TargetPosition : LREAL
GET // PUBLIC
TargetPosition := axis_ref.NcToPlc.TargetPos;
END_GET
END_PROPERTY

END_FUNCTION_BLOCK

// ---- Functions/Mc2EncoderReferenceModeConvertFrom.TcPOU
FUNCTION Mc2EncoderReferenceModeConvertFrom : EncoderReferenceMode
VAR_INPUT
	encoder_reference_mode : Tc2_Mc2.E_EncoderReferenceMode;
END_VAR

CASE encoder_reference_mode OF
    EncoderReferenceMode_Default: Mc2EncoderReferenceModeConvertFrom := EncoderReferenceMode.Default;
    EncoderReferenceMode_PlcCam: Mc2EncoderReferenceModeConvertFrom := EncoderReferenceMode.PlcCam;
    EncoderReferenceMode_HardwareSync: Mc2EncoderReferenceModeConvertFrom := EncoderReferenceMode.HardwareSync;
    EncoderReferenceMode_HardwareLatchPos: Mc2EncoderReferenceModeConvertFrom := EncoderReferenceMode.HardwareLatchPositive;
    EncoderReferenceMode_HardwareLatchNeg: Mc2EncoderReferenceModeConvertFrom := EncoderReferenceMode.HardwareLatchNegative;
    EncoderReferenceMode_SoftwareSync: Mc2EncoderReferenceModeConvertFrom := EncoderReferenceMode.SoftwareSync;
    EncoderReferenceMode_SoftDriveLatchPos: Mc2EncoderReferenceModeConvertFrom := EncoderReferenceMode.SoftDriveLatchPositive;
    EncoderReferenceMode_SoftDriveLatchNeg: Mc2EncoderReferenceModeConvertFrom := EncoderReferenceMode.SoftDriveLatchNegative;
END_CASE

END_FUNCTION

// ---- Functions/Mc2EncoderReferenceModeConvertTo.TcPOU
FUNCTION Mc2EncoderReferenceModeConvertTo : Tc2_Mc2.E_EncoderReferenceMode
VAR_INPUT
	encoder_reference_mode : EncoderReferenceMode;
END_VAR

CASE encoder_reference_mode OF
    EncoderReferenceMode.Default: Mc2EncoderReferenceModeConvertTo := EncoderReferenceMode_Default;
    EncoderReferenceMode.PlcCam: Mc2EncoderReferenceModeConvertTo := EncoderReferenceMode_PlcCam;
    EncoderReferenceMode.HardwareSync: Mc2EncoderReferenceModeConvertTo := EncoderReferenceMode_HardwareSync;
    EncoderReferenceMode.HardwareLatchPositive: Mc2EncoderReferenceModeConvertTo := EncoderReferenceMode_HardwareLatchPos;
    EncoderReferenceMode.HardwareLatchNegative: Mc2EncoderReferenceModeConvertTo := EncoderReferenceMode_HardwareLatchNeg;
    EncoderReferenceMode.SoftwareSync: Mc2EncoderReferenceModeConvertTo := EncoderReferenceMode_SoftwareSync;
    EncoderReferenceMode.SoftDriveLatchPositive: Mc2EncoderReferenceModeConvertTo := EncoderReferenceMode_SoftDriveLatchPos;
    EncoderReferenceMode.SoftDriveLatchNegative: Mc2EncoderReferenceModeConvertTo := EncoderReferenceMode_SoftDriveLatchNeg;
END_CASE

END_FUNCTION

// ---- Functions/Mc2HomingModeConvertFrom.TcPOU
FUNCTION Mc2HomingModeConvertFrom : HomingMode
VAR_INPUT
	homing_mode : Tc2_Mc2.Mc_HomingMode;
END_VAR

CASE homing_mode OF
	Tc2_Mc2.MC_DefaultHoming: Mc2HomingModeConvertFrom := HomingMode.DefaultHoming;
	Tc2_Mc2.MC_Direct: Mc2HomingModeConvertFrom := HomingMode.Direct;
	Tc2_Mc2.MC_ForceCalibration: Mc2HomingModeConvertFrom := HomingMode.ForceCalibration;
	Tc2_Mc2.MC_ResetCalibration: Mc2HomingModeConvertFrom := HomingMode.ResetCalibration;
END_CASE

END_FUNCTION
